LIN {X 0,Y 460.804,Z 363.083,A -85,B 0,C 180,E1 -7827.377,E2 -7827.377} C_VEL
LIN {X 0,Y 460.857,Z 363.08,A -85,B 0,C 180,E1 -7830,E2 -7830} C_VEL
LIN {X 0,Y 460.828,Z 363.084,A -85,B 0,C 180,E1 -7832.622,E2 -7832.622} C_VEL
LIN {X 0,Y 460.706,Z 363.1,A -85,B 0,C 180,E1 -7836.13,E2 -7836.13} C_VEL
LIN {X 0,Y 460.632,Z 363.104,A -85,B 0,C 180,E1 -7838.776,E2 -7838.776} C_VEL
LIN {X 0,Y 460.617,Z 363.109,A -85,B 0,C 180,E1 -7842.445,E2 -7842.445} C_VEL
LIN {X 0,Y 460.604,Z 363.112,A -85,B 0,C 180,E1 -7845.997,E2 -7845.997} C_VEL
LIN {X 0,Y 460.575,Z 363.112,A -85,B 0,C 180,E1 -7848.902,E2 -7848.902} C_VEL
LIN {X 0,Y 460.519,Z 363.124,A -85,B 0,C 180,E1 -7851.485,E2 -7851.485} C_VEL
LIN {X 0,Y 460.545,Z 363.119,A -85,B 0,C 180,E1 -7854.332,E2 -7854.332} C_VEL
LIN {X 0,Y 460.583,Z 363.112,A -85,B 0,C 180,E1 -7857.243,E2 -7857.243} C_VEL
LIN {X 0,Y 460.514,Z 363.119,A -85,B 0,C 180,E1 -7860.24,E2 -7860.24} C_VEL
LIN {X 0,Y 460.532,Z 363.121,A -85,B 0,C 180,E1 -7863.325,E2 -7863.325} C_VEL
LIN {X 0,Y 460.479,Z 363.127,A -85,B 0,C 180,E1 -7866.529,E2 -7866.529} C_VEL
LIN {X 0,Y 460.561,Z 363.116,A -85,B 0,C 180,E1 -7869.859,E2 -7869.859} C_VEL
LIN {X 0,Y 460.516,Z 363.122,A -85,B 0,C 180,E1 -7872.9,E2 -7872.9} C_VEL
LIN {X 0,Y 460.514,Z 363.122,A -85,B 0,C 180,E1 -7875.83,E2 -7875.83} C_VEL
LIN {X 0,Y 460.533,Z 363.119,A -85,B 0,C 180,E1 -7878.989,E2 -7878.989} C_VEL
LIN {X 0,Y 460.529,Z 363.123,A -85,B 0,C 180,E1 -7881.267,E2 -7881.267} C_VEL
LIN {X 0,Y 460.513,Z 363.122,A -85,B 0,C 180,E1 -7884.554,E2 -7884.554} C_VEL
LIN {X 0,Y 460.534,Z 363.12,A -85,B 0,C 180,E1 -7887.716,E2 -7887.716} C_VEL
LIN {X 0,Y 460.543,Z 363.118,A -85,B 0,C 180,E1 -7890.769,E2 -7890.769} C_VEL
LIN {X 0,Y 460.566,Z 363.112,A -85,B 0,C 180,E1 -7893.735,E2 -7893.735} C_VEL
LIN {X 0,Y 460.549,Z 363.12,A -85,B 0,C 180,E1 -7896.624,E2 -7896.624} C_VEL
LIN {X 0,Y 460.555,Z 363.118,A -85,B 0,C 180,E1 -7899.453,E2 -7899.453} C_VEL
LIN {X 0,Y 460.562,Z 363.114,A -85,B 0,C 180,E1 -7902.23,E2 -7902.23} C_VEL
LIN {X 0,Y 460.568,Z 363.116,A -85,B 0,C 180,E1 -7904.965,E2 -7904.965} C_VEL
LIN {X 0,Y 460.633,Z 363.106,A -85,B 0,C 180,E1 -7907.666,E2 -7907.666} C_VEL
LIN {X 0,Y 460.632,Z 363.109,A -85,B 0,C 180,E1 -7911.224,E2 -7911.224} C_VEL
LIN {X 0,Y 460.713,Z 363.095,A -85,B 0,C 180,E1 -7913.87,E2 -7913.87} C_VEL
LIN {X 0,Y 460.803,Z 363.084,A -85,B 0,C 180,E1 -7917.377,E2 -7917.377} C_VEL
LIN {X 0,Y 460.857,Z 363.081,A -85,B 0,C 180,E1 -7920,E2 -7920} C_VEL
LIN {X 0,Y 460.827,Z 363.083,A -85,B 0,C 180,E1 -7922.622,E2 -7922.622} C_VEL
LIN {X 0,Y 460.712,Z 363.097,A -85,B 0,C 180,E1 -7926.13,E2 -7926.13} C_VEL
LIN {X 0,Y 460.631,Z 363.106,A -85,B 0,C 180,E1 -7928.776,E2 -7928.776} C_VEL
LIN {X 0,Y 460.616,Z 363.109,A -85,B 0,C 180,E1 -7932.445,E2 -7932.445} C_VEL
LIN {X 0,Y 460.602,Z 363.11,A -85,B 0,C 180,E1 -7935.997,E2 -7935.997} C_VEL
LIN {X 0,Y 460.571,Z 363.114,A -85,B 0,C 180,E1 -7939.615,E2 -7939.615} C_VEL
LIN {X 0,Y 460.513,Z 363.121,A -85,B 0,C 180,E1 -7942.429,E2 -7942.429} C_VEL
LIN {X 0,Y 460.57,Z 363.114,A -85,B 0,C 180,E1 -7945.802,E2 -7945.802} C_VEL
LIN {X 0,Y 460.554,Z 363.118,A -85,B 0,C 180,E1 -7948.233,E2 -7948.233} C_VEL
LIN {X 0,Y 460.523,Z 363.12,A -85,B 0,C 180,E1 -7951.283,E2 -7951.283} C_VEL
LIN {X 0,Y 460.536,Z 363.121,A -85,B 0,C 180,E1 -7954.506,E2 -7954.506} C_VEL
LIN {X 0,Y 460.53,Z 363.119,A -85,B 0,C 180,E1 -7957.62,E2 -7957.62} C_VEL
LIN {X 0,Y 460.545,Z 363.117,A -85,B 0,C 180,E1 -7960.27,E2 -7960.27} C_VEL
LIN {X 0,Y 460.511,Z 363.125,A -85,B 0,C 180,E1 -7963.374,E2 -7963.374} C_VEL
LIN {X 0,Y 460.511,Z 363.122,A -85,B 0,C 180,E1 -7966.626,E2 -7966.626} C_VEL
LIN {X 0,Y 460.542,Z 363.121,A -85,B 0,C 180,E1 -7969.731,E2 -7969.731} C_VEL
LIN {X 0,Y 460.501,Z 363.121,A -85,B 0,C 180,E1 -7972.524,E2 -7972.524} C_VEL
LIN {X 0,Y 460.548,Z 363.115,A -85,B 0,C 180,E1 -7975.624,E2 -7975.624} C_VEL
LIN {X 0,Y 460.613,Z 363.263,A -85,B 0,C 180,E1 -7976.739,E2 -7976.739} C_VEL
LIN {X 0,Y 463.241,Z 375.686,A -85,B 0,C 180,E1 -7979.857,E2 -7979.857} C_VEL
LIN {X 0,Y 464.177,Z 380.491,A -85,B 0,C 180,E1 -7981.02,E2 -7981.02} C_VEL
LIN {X 0,Y 463.73,Z 388.112,A -85,B 0,C 180,E1 -7982.713,E2 -7982.713} C_VEL
LIN {X 0,Y 462.742,Z 402.3,A -85,B 0,C 180,E1 -7985.791,E2 -7985.791} C_VEL
LIN {X 0,Y 461.732,Z 418.733,A -85,B 0,C 180,E1 -7989.275,E2 -7989.275} C_VEL
LIN {X 0,Y 461.049,Z 434.161,A -85,B 0,C 180,E1 -7992.479,E2 -7992.479} C_VEL
LIN {X 0,Y 460.614,Z 445.332,A -85,B 0,C 180,E1 -7994.768,E2 -7994.768} C_VEL
LIN {X 0,Y 462.065,Z 459.581,A -85,B 0,C 180,E1 -7995.156,E2 -7995.156} C_VEL
LIN {X 0,Y 462.428,Z 464.556,A -85,B 0,C 180,E1 -7995.336,E2 -7995.336} C_VEL
LIN {X 0,Y 462.148,Z 476.548,A -85,B 0,C 180,E1 -7995.862,E2 -7995.862} C_VEL
LIN {X 0,Y 461.723,Z 488.674,A -85,B 0,C 180,E1 -7996.578,E2 -7996.578} C_VEL
LIN {X 0,Y 461.341,Z 499.812,A -85,B 0,C 180,E1 -7997.428,E2 -7997.428} C_VEL
LIN {X 0,Y 460.794,Z 510.557,A -85,B 0,C 180,E1 -7998.452,E2 -7998.452} C_VEL
LIN {X 0,Y 460.459,Z 519.001,A -85,B 0,C 180,E1 -7999.446,E2 -7999.446} C_VEL
LIN {X 0,Y 460.111,Z 528.13,A -85,B 0,C 180,E1 -8000.771,E2 -8000.771} C_VEL
LIN {X 0,Y 459.892,Z 535.454,A -85,B 0,C 180,E1 -8002.095,E2 -8002.095} C_VEL
LIN {X 0,Y 459.735,Z 541.743,A -85,B 0,C 180,E1 -8003.546,E2 -8003.546} C_VEL
LIN {X 0,Y 459.728,Z 545.798,A -85,B 0,C 180,E1 -8004.737,E2 -8004.737} C_VEL
LIN {X 0,Y 459.681,Z 548.168,A -85,B 0,C 180,E1 -8005.616,E2 -8005.616} C_VEL
LIN {X 0,Y 459.745,Z 550.103,A -85,B 0,C 180,E1 -8006.494,E2 -8006.494} C_VEL
LIN {X 0,Y 459.762,Z 551.576,A -85,B 0,C 180,E1 -8007.372,E2 -8007.372} C_VEL
LIN {X 0,Y 459.6,Z 553.186,A -85,B 0,C 180,E1 -8009.124,E2 -8009.124} C_VEL
LIN {X 0,Y 459.605,Z 553.392,A -85,B 0,C 180,E1 -8010,E2 -8010} C_VEL
LIN {X 0,Y 459.603,Z 553.142,A -85,B 0,C 180,E1 -8010.876,E2 -8010.876} C_VEL
LIN {X 0,Y 459.765,Z 551.428,A -85,B 0,C 180,E1 -8012.628,E2 -8012.628} C_VEL
LIN {X 0,Y 459.759,Z 549.92,A -85,B 0,C 180,E1 -8013.506,E2 -8013.506} C_VEL
LIN {X 0,Y 459.668,Z 546.785,A -85,B 0,C 180,E1 -8014.824,E2 -8014.824} C_VEL
LIN {X 0,Y 459.757,Z 542.559,A -85,B 0,C 180,E1 -8016.143,E2 -8016.143} C_VEL
LIN {X 0,Y 459.854,Z 537.104,A -85,B 0,C 180,E1 -8017.464,E2 -8017.464} C_VEL
LIN {X 0,Y 460.018,Z 530.243,A -85,B 0,C 180,E1 -8018.788,E2 -8018.788} C_VEL
LIN {X 0,Y 460.303,Z 521.708,A -85,B 0,C 180,E1 -8020.113,E2 -8020.113} C_VEL
LIN {X 0,Y 460.698,Z 512.901,A -85,B 0,C 180,E1 -8021.216,E2 -8021.216} C_VEL
LIN {X 0,Y 461.092,Z 503.223,A -85,B 0,C 180,E1 -8022.209,E2 -8022.209} C_VEL
LIN {X 0,Y 461.542,Z 492.388,A -85,B 0,C 180,E1 -8023.112,E2 -8023.112} C_VEL
LIN {X 0,Y 461.963,Z 480.948,A -85,B 0,C 180,E1 -8023.864,E2 -8023.864} C_VEL
LIN {X 0,Y 462.412,Z 467.554,A -85,B 0,C 180,E1 -8024.524,E2 -8024.524} C_VEL
LIN {X 0,Y 462.324,Z 461.772,A -85,B 0,C 180,E1 -8024.751,E2 -8024.751} C_VEL
LIN {X 0,Y 461.146,Z 449.381,A -85,B 0,C 180,E1 -8025.143,E2 -8025.143} C_VEL
LIN {X 0,Y 460.603,Z 444.609,A -85,B 0,C 180,E1 -8025.26,E2 -8025.26} C_VEL
LIN {X 0,Y 461.149,Z 429.066,A -85,B 0,C 180,E1 -8028.435,E2 -8028.435} C_VEL
LIN {X 0,Y 461.893,Z 415.007,A -85,B 0,C 180,E1 -8031.419,E2 -8031.419} C_VEL
LIN {X 0,Y 462.96,Z 400.561,A -85,B 0,C 180,E1 -8034.674,E2 -8034.674} C_VEL
LIN {X 0,Y 464.43,Z 386.973,A -85,B 0,C 180,E1 -8037.977,E2 -8037.977} C_VEL
LIN {X 0,Y 464.771,Z 383.328,A -85,B 0,C 180,E1 -8038.94,E2 -8038.94} C_VEL
LIN {X 0,Y 463.986,Z 377.841,A -85,B 0,C 180,E1 -8040.594,E2 -8040.594} C_VEL
LIN {X 0,Y 462.269,Z 370.242,A -85,B 0,C 180,E1 -8043.261,E2 -8043.261} C_VEL
LIN {X 0,Y 461.021,Z 365.258,A -85,B 0,C 180,E1 -8045.401,E2 -8045.401} C_VEL
LIN {X 0,Y 460.479,Z 363.13,A -85,B 0,C 180,E1 -8046.529,E2 -8046.529} C_VEL
LIN {X 0,Y 460.535,Z 363.121,A -85,B 0,C 180,E1 -8049.862,E2 -8049.862} C_VEL
LIN {X 0,Y 460.52,Z 363.124,A -85,B 0,C 180,E1 -8052.901,E2 -8052.901} C_VEL
LIN {X 0,Y 460.522,Z 363.123,A -85,B 0,C 180,E1 -8055.829,E2 -8055.829} C_VEL
LIN {X 0,Y 460.544,Z 363.12,A -85,B 0,C 180,E1 -8058.99,E2 -8058.99} C_VEL
LIN {X 0,Y 460.55,Z 363.12,A -85,B 0,C 180,E1 -8061.269,E2 -8061.269} C_VEL
LIN {X 0,Y 460.516,Z 363.125,A -85,B 0,C 180,E1 -8064.555,E2 -8064.555} C_VEL
LIN {X 0,Y 460.57,Z 363.243,A -85,B 0,C 180,E1 -8065.626,E2 -8065.626} C_VEL
LIN {X 0,Y 461.132,Z 366.331,A -85,B 0,C 180,E1 -8067.763,E2 -8067.763} C_VEL
LIN {X 0,Y 461.472,Z 370.302,A -85,B 0,C 180,E1 -8070.237,E2 -8070.237} C_VEL
LIN {X 0,Y 461.266,Z 374.775,A -85,B 0,C 180,E1 -8072.8,E2 -8072.8} C_VEL
LIN {X 0,Y 460.953,Z 380,A -85,B 0,C 180,E1 -8075.691,E2 -8075.691} C_VEL
LIN {X 0,Y 460.78,Z 385.295,A -85,B 0,C 180,E1 -8078.527,E2 -8078.527} C_VEL
LIN {X 0,Y 460.589,Z 390.661,A -85,B 0,C 180,E1 -8081.311,E2 -8081.311} C_VEL
LIN {X 0,Y 460.395,Z 396.113,A -85,B 0,C 180,E1 -8084.093,E2 -8084.093} C_VEL
LIN {X 0,Y 460.212,Z 403.49,A -85,B 0,C 180,E1 -8087.786,E2 -8087.786} C_VEL
LIN {X 0,Y 460.028,Z 408.741,A -85,B 0,C 180,E1 -8090.353,E2 -8090.353} C_VEL
LIN {X 0,Y 461.717,Z 418.634,A -85,B 0,C 180,E1 -8090.914,E2 -8090.914} C_VEL
LIN {X 0,Y 461.425,Z 428.414,A -85,B 0,C 180,E1 -8091.57,E2 -8091.57} C_VEL
LIN {X 0,Y 461.114,Z 437.441,A -85,B 0,C 180,E1 -8092.382,E2 -8092.382} C_VEL
LIN {X 0,Y 460.834,Z 444.616,A -85,B 0,C 180,E1 -8093.212,E2 -8093.212} C_VEL
LIN {X 0,Y 460.601,Z 450.612,A -85,B 0,C 180,E1 -8094.088,E2 -8094.088} C_VEL
LIN {X 0,Y 460.341,Z 456.412,A -85,B 0,C 180,E1 -8095.183,E2 -8095.183} C_VEL
LIN {X 0,Y 460.304,Z 459.937,A -85,B 0,C 180,E1 -8096.06,E2 -8096.06} C_VEL
LIN {X 0,Y 460.105,Z 462.654,A -85,B 0,C 180,E1 -8096.935,E2 -8096.935} C_VEL
LIN {X 0,Y 459.887,Z 463.739,A -85,B 0,C 180,E1 -8097.372,E2 -8097.372} C_VEL
LIN {X 0,Y 459.78,Z 465.333,A -85,B 0,C 180,E1 -8098.248,E2 -8098.248} C_VEL
LIN {X 0,Y 459.732,Z 466.235,A -85,B 0,C 180,E1 -8099.124,E2 -8099.124} C_VEL
LIN {X 0,Y 459.71,Z 466.468,A -85,B 0,C 180,E1 -8100,E2 -8100} C_VEL
LIN {X 0,Y 459.703,Z 466.034,A -85,B 0,C 180,E1 -8100.876,E2 -8100.876} C_VEL
LIN {X 0,Y 459.727,Z 464.929,A -85,B 0,C 180,E1 -8101.752,E2 -8101.752} C_VEL
LIN {X 0,Y 460.036,Z 461.941,A -85,B 0,C 180,E1 -8103.065,E2 -8103.065} C_VEL
LIN {X 0,Y 460.22,Z 457.216,A -85,B 0,C 180,E1 -8104.379,E2 -8104.379} C_VEL
LIN {X 0,Y 460.371,Z 451.718,A -85,B 0,C 180,E1 -8105.475,E2 -8105.475} C_VEL
LIN {X 0,Y 460.495,Z 446.043,A -85,B 0,C 180,E1 -8106.353,E2 -8106.353} C_VEL
LIN {X 0,Y 460.645,Z 438.702,A -85,B 0,C 180,E1 -8107.247,E2 -8107.247} C_VEL
LIN {X 0,Y 460.944,Z 429.462,A -85,B 0,C 180,E1 -8108.108,E2 -8108.108} C_VEL
LIN {X 0,Y 461.224,Z 420.011,A -85,B 0,C 180,E1 -8108.765,E2 -8108.765} C_VEL
LIN {X 0,Y 461.037,Z 415.021,A -85,B 0,C 180,E1 -8109.045,E2 -8109.045} C_VEL
LIN {X 0,Y 459.779,Z 406.698,A -85,B 0,C 180,E1 -8109.458,E2 -8109.458} C_VEL
LIN {X 0,Y 459.856,Z 400.472,A -85,B 0,C 180,E1 -8112.355,E2 -8112.355} C_VEL
LIN {X 0,Y 460.013,Z 392.824,A -85,B 0,C 180,E1 -8115.962,E2 -8115.962} C_VEL
LIN {X 0,Y 460.143,Z 387.009,A -85,B 0,C 180,E1 -8118.744,E2 -8118.744} C_VEL
LIN {X 0,Y 460.21,Z 381.312,A -85,B 0,C 180,E1 -8121.501,E2 -8121.501} C_VEL
LIN {X 0,Y 460.342,Z 375.512,A -85,B 0,C 180,E1 -8124.344,E2 -8124.344} C_VEL
LIN {X 0,Y 460.491,Z 369.662,A -85,B 0,C 180,E1 -8127.249,E2 -8127.249} C_VEL
LIN {X 0,Y 460.777,Z 363.737,A -85,B 0,C 180,E1 -8130.221,E2 -8130.221} C_VEL
LIN {X 0,Y 460.664,Z 363.105,A -85,B 0,C 180,E1 -8130.609,E2 -8130.609} C_VEL
LIN {X 0,Y 460.552,Z 363.117,A -85,B 0,C 180,E1 -8134.376,E2 -8134.376} C_VEL
LIN {X 0,Y 460.532,Z 363.12,A -85,B 0,C 180,E1 -8137.621,E2 -8137.621} C_VEL
LIN {X 0,Y 460.545,Z 363.117,A -85,B 0,C 180,E1 -8140.269,E2 -8140.269} C_VEL
LIN {X 0,Y 460.503,Z 363.121,A -85,B 0,C 180,E1 -8143.375,E2 -8143.375} C_VEL
LIN {X 0,Y 460.512,Z 363.123,A -85,B 0,C 180,E1 -8146.626,E2 -8146.626} C_VEL
LIN {X 0,Y 460.546,Z 363.118,A -85,B 0,C 180,E1 -8149.73,E2 -8149.73} C_VEL
LIN {X 0,Y 460.503,Z 363.123,A -85,B 0,C 180,E1 -8152.524,E2 -8152.524} C_VEL
LIN {X 0,Y 460.549,Z 363.115,A -85,B 0,C 180,E1 -8155.624,E2 -8155.624} C_VEL
LIN {X 0,Y 460.541,Z 363.118,A -85,B 0,C 180,E1 -8158.745,E2 -8158.745} C_VEL
LIN {X 0,Y 460.592,Z 363.111,A -85,B 0,C 180,E1 -8162.252,E2 -8162.252} C_VEL
LIN {X 0,Y 460.535,Z 363.116,A -85,B 0,C 180,E1 -8165.667,E2 -8165.667} C_VEL
LIN {X 0,Y 460.525,Z 363.12,A -85,B 0,C 180,E1 -8168.578,E2 -8168.578} C_VEL
LIN {X 0,Y 460.594,Z 363.112,A -85,B 0,C 180,E1 -8171.311,E2 -8171.311} C_VEL
LIN {X 0,Y 460.571,Z 363.112,A -85,B 0,C 180,E1 -8174.586,E2 -8174.586} C_VEL
LIN {X 0,Y 460.613,Z 363.108,A -85,B 0,C 180,E1 -8177.666,E2 -8177.666} C_VEL
LIN {X 0,Y 460.606,Z 363.108,A -85,B 0,C 180,E1 -8178.39,E2 -8178.39} C_VEL
LIN {X 0,Y 459.966,Z 363.191,A -85,B 0,C 180,E1 -8179.12,E2 -8179.12} C_VEL
LIN {X 0,Y 457.128,Z 363.545,A -85,B 0,C 180,E1 -8180.306,E2 -8180.306} C_VEL
LIN {X 0,Y 454.734,Z 363.842,A -85,B 0,C 180,E1 -8181.262,E2 -8181.262} C_VEL
LIN {X 0,Y 453.735,Z 363.966,A -85,B 0,C 180,E1 -8182.001,E2 -8182.001} C_VEL
LIN {X 0,Y 453.671,Z 363.974,A -85,B 0,C 180,E1 -8182.251,E2 -8182.251} C_VEL
LIN {X 0,Y 453.672,Z 363.975,A -85,B 0,C 180,E1 -8184.667,E2 -8184.667} C_VEL
LIN {X 0,Y 453.748,Z 363.962,A -85,B 0,C 180,E1 -8187.337,E2 -8187.337} C_VEL
LIN {X 0,Y 453.827,Z 363.956,A -85,B 0,C 180,E1 -8190,E2 -8190} C_VEL
LIN {X 0,Y 453.769,Z 363.963,A -85,B 0,C 180,E1 -8192.663,E2 -8192.663} C_VEL
LIN {X 0,Y 453.673,Z 363.976,A -85,B 0,C 180,E1 -8196.225,E2 -8196.225} C_VEL
LIN {X 0,Y 453.596,Z 363.98,A -85,B 0,C 180,E1 -8198.913,E2 -8198.913} C_VEL
LIN {X 0,Y 453.567,Z 363.987,A -85,B 0,C 180,E1 -8202.529,E2 -8202.529} C_VEL
LIN {X 0,Y 453.548,Z 363.991,A -85,B 0,C 180,E1 -8206.196,E2 -8206.196} C_VEL
LIN {X 0,Y 453.524,Z 363.99,A -85,B 0,C 180,E1 -8209.041,E2 -8209.041} C_VEL
LIN {X 0,Y 453.48,Z 363.998,A -85,B 0,C 180,E1 -8211.836,E2 -8211.836} C_VEL
LIN {X 0,Y 453.517,Z 363.994,A -85,B 0,C 180,E1 -8214.734,E2 -8214.734} C_VEL
LIN {X 0,Y 453.541,Z 363.992,A -85,B 0,C 180,E1 -8217.961,E2 -8217.961} C_VEL
LIN {X 0,Y 453.469,Z 364.001,A -85,B 0,C 180,E1 -8221.525,E2 -8221.525} C_VEL
LIN {X 0,Y 453.49,Z 363.997,A -85,B 0,C 180,E1 -8224.777,E2 -8224.777} C_VEL
LIN {X 0,Y 453.467,Z 363.999,A -85,B 0,C 180,E1 -8228.311,E2 -8228.311} C_VEL
LIN {X 0,Y 453.497,Z 363.994,A -85,B 0,C 180,E1 -8230.609,E2 -8230.609} C_VEL
LIN {X 0,Y 453.459,Z 364.003,A -85,B 0,C 180,E1 -8233.244,E2 -8233.244} C_VEL
LIN {X 0,Y 453.469,Z 363.999,A -85,B 0,C 180,E1 -8235.779,E2 -8235.779} C_VEL
LIN {X 0,Y 453.481,Z 363.998,A -85,B 0,C 180,E1 -8238.209,E2 -8238.209} C_VEL
LIN {X 0,Y 453.497,Z 363.995,A -85,B 0,C 180,E1 -8240.793,E2 -8240.793} C_VEL
LIN {X 0,Y 453.457,Z 363.999,A -85,B 0,C 180,E1 -8243.917,E2 -8243.917} C_VEL
LIN {X 0,Y 453.485,Z 363.997,A -85,B 0,C 180,E1 -8247.151,E2 -8247.151} C_VEL
LIN {X 0,Y 453.478,Z 363.998,A -85,B 0,C 180,E1 -8250.268,E2 -8250.268} C_VEL
LIN {X 0,Y 453.509,Z 363.994,A -85,B 0,C 180,E1 -8253.294,E2 -8253.294} C_VEL
LIN {X 0,Y 453.507,Z 363.994,A -85,B 0,C 180,E1 -8256.239,E2 -8256.239} C_VEL
LIN {X 0,Y 453.486,Z 363.997,A -85,B 0,C 180,E1 -8259.118,E2 -8259.118} C_VEL
LIN {X 0,Y 453.515,Z 363.993,A -85,B 0,C 180,E1 -8261.945,E2 -8261.945} C_VEL
LIN {X 0,Y 453.543,Z 363.993,A -85,B 0,C 180,E1 -8264.726,E2 -8264.726} C_VEL
LIN {X 0,Y 453.605,Z 363.982,A -85,B 0,C 180,E1 -8267.472,E2 -8267.472} C_VEL
LIN {X 0,Y 453.596,Z 363.985,A -85,B 0,C 180,E1 -8271.087,E2 -8271.087} C_VEL
LIN {X 0,Y 453.68,Z 363.972,A -85,B 0,C 180,E1 -8273.775,E2 -8273.775} C_VEL
LIN {X 0,Y 453.747,Z 363.963,A -85,B 0,C 180,E1 -8277.337,E2 -8277.337} C_VEL
LIN {X 0,Y 453.827,Z 363.957,A -85,B 0,C 180,E1 -8280,E2 -8280} C_VEL
LIN {X 0,Y 453.768,Z 363.963,A -85,B 0,C 180,E1 -8282.663,E2 -8282.663} C_VEL
LIN {X 0,Y 453.68,Z 363.974,A -85,B 0,C 180,E1 -8286.225,E2 -8286.225} C_VEL
LIN {X 0,Y 453.594,Z 363.982,A -85,B 0,C 180,E1 -8288.913,E2 -8288.913} C_VEL
LIN {X 0,Y 453.566,Z 363.987,A -85,B 0,C 180,E1 -8292.529,E2 -8292.529} C_VEL
LIN {X 0,Y 453.546,Z 363.991,A -85,B 0,C 180,E1 -8296.196,E2 -8296.196} C_VEL
LIN {X 0,Y 453.52,Z 363.991,A -85,B 0,C 180,E1 -8299.04,E2 -8299.04} C_VEL
LIN {X 0,Y 453.478,Z 364,A -85,B 0,C 180,E1 -8301.836,E2 -8301.836} C_VEL
LIN {X 0,Y 453.515,Z 363.994,A -85,B 0,C 180,E1 -8304.734,E2 -8304.734} C_VEL
LIN {X 0,Y 453.534,Z 363.993,A -85,B 0,C 180,E1 -8307.96,E2 -8307.96} C_VEL
LIN {X 0,Y 453.468,Z 364.001,A -85,B 0,C 180,E1 -8311.525,E2 -8311.525} C_VEL
LIN {X 0,Y 453.491,Z 363.997,A -85,B 0,C 180,E1 -8314.778,E2 -8314.778} C_VEL
LIN {X 0,Y 453.475,Z 363.999,A -85,B 0,C 180,E1 -8318.311,E2 -8318.311} C_VEL
LIN {X 0,Y 453.496,Z 363.993,A -85,B 0,C 180,E1 -8320.609,E2 -8320.609} C_VEL
LIN {X 0,Y 453.465,Z 364.001,A -85,B 0,C 180,E1 -8323.245,E2 -8323.245} C_VEL
LIN {X 0,Y 453.475,Z 363.998,A -85,B 0,C 180,E1 -8325.78,E2 -8325.78} C_VEL
LIN {X 0,Y 453.484,Z 363.999,A -85,B 0,C 180,E1 -8328.21,E2 -8328.21} C_VEL
LIN {X 0,Y 453.489,Z 363.992,A -85,B 0,C 180,E1 -8330.794,E2 -8330.794} C_VEL
LIN {X 0,Y 453.456,Z 364.001,A -85,B 0,C 180,E1 -8333.917,E2 -8333.917} C_VEL
LIN {X 0,Y 453.551,Z 364.167,A -85,B 0,C 180,E1 -8336.43,E2 -8336.43} C_VEL
LIN {X 0,Y 456.236,Z 376.608,A -85,B 0,C 180,E1 -8339.615,E2 -8339.615} C_VEL
LIN {X 0,Y 457.29,Z 382.993,A -85,B 0,C 180,E1 -8341.166,E2 -8341.166} C_VEL
LIN {X 0,Y 456.263,Z 396.521,A -85,B 0,C 180,E1 -8344.205,E2 -8344.205} C_VEL
LIN {X 0,Y 455.153,Z 412.385,A -85,B 0,C 180,E1 -8347.665,E2 -8347.665} C_VEL
LIN {X 0,Y 454.34,Z 426.401,A -85,B 0,C 180,E1 -8350.663,E2 -8350.663} C_VEL
LIN {X 0,Y 453.726,Z 440.257,A -85,B 0,C 180,E1 -8353.58,E2 -8353.58} C_VEL
LIN {X 0,Y 453.581,Z 445.076,A -85,B 0,C 180,E1 -8354.585,E2 -8354.585} C_VEL
LIN {X 0,Y 454.967,Z 459.21,A -85,B 0,C 180,E1 -8354.976,E2 -8354.976} C_VEL
LIN {X 0,Y 455.443,Z 464.957,A -85,B 0,C 180,E1 -8355.192,E2 -8355.192} C_VEL
LIN {X 0,Y 455.135,Z 477.261,A -85,B 0,C 180,E1 -8355.753,E2 -8355.753} C_VEL
LIN {X 0,Y 454.693,Z 489.054,A -85,B 0,C 180,E1 -8356.48,E2 -8356.48} C_VEL
LIN {X 0,Y 454.283,Z 500.104,A -85,B 0,C 180,E1 -8357.35,E2 -8357.35} C_VEL
LIN {X 0,Y 453.732,Z 510.602,A -85,B 0,C 180,E1 -8358.383,E2 -8358.383} C_VEL
LIN {X 0,Y 453.326,Z 519.758,A -85,B 0,C 180,E1 -8359.504,E2 -8359.504} C_VEL
LIN {X 0,Y 453.015,Z 528.665,A -85,B 0,C 180,E1 -8360.85,E2 -8360.85} C_VEL
LIN {X 0,Y 452.805,Z 535.733,A -85,B 0,C 180,E1 -8362.195,E2 -8362.195} C_VEL
LIN {X 0,Y 452.65,Z 541.426,A -85,B 0,C 180,E1 -8363.559,E2 -8363.559} C_VEL
LIN {X 0,Y 452.589,Z 546.336,A -85,B 0,C 180,E1 -8365.101,E2 -8365.101} C_VEL
LIN {X 0,Y 452.674,Z 549.413,A -85,B 0,C 180,E1 -8366.44,E2 -8366.44} C_VEL
LIN {X 0,Y 452.706,Z 550.901,A -85,B 0,C 180,E1 -8367.331,E2 -8367.331} C_VEL
LIN {X 0,Y 452.589,Z 551.908,A -85,B 0,C 180,E1 -8368.22,E2 -8368.22} C_VEL
LIN {X 0,Y 452.533,Z 552.516,A -85,B 0,C 180,E1 -8369.11,E2 -8369.11} C_VEL
LIN {X 0,Y 452.536,Z 552.724,A -85,B 0,C 180,E1 -8370,E2 -8370} C_VEL
LIN {X 0,Y 452.536,Z 552.477,A -85,B 0,C 180,E1 -8370.89,E2 -8370.89} C_VEL
LIN {X 0,Y 452.592,Z 551.819,A -85,B 0,C 180,E1 -8371.78,E2 -8371.78} C_VEL
LIN {X 0,Y 452.71,Z 550.759,A -85,B 0,C 180,E1 -8372.669,E2 -8372.669} C_VEL
LIN {X 0,Y 452.654,Z 548.304,A -85,B 0,C 180,E1 -8374.006,E2 -8374.006} C_VEL
LIN {X 0,Y 452.677,Z 544.812,A -85,B 0,C 180,E1 -8375.345,E2 -8375.345} C_VEL
LIN {X 0,Y 452.759,Z 539.621,A -85,B 0,C 180,E1 -8376.832,E2 -8376.832} C_VEL
LIN {X 0,Y 452.882,Z 533.154,A -85,B 0,C 180,E1 -8378.253,E2 -8378.253} C_VEL
LIN {X 0,Y 453.099,Z 525.487,A -85,B 0,C 180,E1 -8379.599,E2 -8379.599} C_VEL
LIN {X 0,Y 453.419,Z 517.654,A -85,B 0,C 180,E1 -8380.72,E2 -8380.72} C_VEL
LIN {X 0,Y 453.861,Z 506.991,A -85,B 0,C 180,E1 -8381.953,E2 -8381.953} C_VEL
LIN {X 0,Y 454.307,Z 496.361,A -85,B 0,C 180,E1 -8382.942,E2 -8382.942} C_VEL
LIN {X 0,Y 454.763,Z 485.534,A -85,B 0,C 180,E1 -8383.746,E2 -8383.746} C_VEL
LIN {X 0,Y 455.326,Z 472.817,A -85,B 0,C 180,E1 -8384.469,E2 -8384.469} C_VEL
LIN {X 0,Y 455.363,Z 462.344,A -85,B 0,C 180,E1 -8384.925,E2 -8384.925} C_VEL
LIN {X 0,Y 454.227,Z 449.851,A -85,B 0,C 180,E1 -8385.347,E2 -8385.347} C_VEL
LIN {X 0,Y 453.567,Z 444.274,A -85,B 0,C 180,E1 -8385.495,E2 -8385.495} C_VEL
LIN {X 0,Y 454.191,Z 428.804,A -85,B 0,C 180,E1 -8388.728,E2 -8388.728} C_VEL
LIN {X 0,Y 454.998,Z 414.943,A -85,B 0,C 180,E1 -8391.76,E2 -8391.76} C_VEL
LIN {X 0,Y 456.14,Z 400.646,A -85,B 0,C 180,E1 -8395.069,E2 -8395.069} C_VEL
LIN {X 0,Y 457.778,Z 387.378,A -85,B 0,C 180,E1 -8398.42,E2 -8398.42} C_VEL
LIN {X 0,Y 457.886,Z 383.82,A -85,B 0,C 180,E1 -8399.417,E2 -8399.417} C_VEL
LIN {X 0,Y 456.615,Z 377.293,A -85,B 0,C 180,E1 -8401.555,E2 -8401.555} C_VEL
LIN {X 0,Y 455.348,Z 371.453,A -85,B 0,C 180,E1 -8403.755,E2 -8403.755} C_VEL
LIN {X 0,Y 454.054,Z 366.532,A -85,B 0,C 180,E1 -8406.028,E2 -8406.028} C_VEL
LIN {X 0,Y 453.471,Z 364.002,A -85,B 0,C 180,E1 -8407.479,E2 -8407.479} C_VEL
LIN {X 0,Y 453.497,Z 363.998,A -85,B 0,C 180,E1 -8410.609,E2 -8410.609} C_VEL
LIN {X 0,Y 453.466,Z 364.002,A -85,B 0,C 180,E1 -8413.245,E2 -8413.245} C_VEL
LIN {X 0,Y 453.476,Z 364.001,A -85,B 0,C 180,E1 -8415.78,E2 -8415.78} C_VEL
LIN {X 0,Y 453.519,Z 363.995,A -85,B 0,C 180,E1 -8419.406,E2 -8419.406} C_VEL
LIN {X 0,Y 453.481,Z 364.001,A -85,B 0,C 180,E1 -8422.223,E2 -8422.223} C_VEL
LIN {X 0,Y 453.476,Z 364.038,A -85,B 0,C 180,E1 -8424.739,E2 -8424.739} C_VEL
LIN {X 0,Y 454.165,Z 367.303,A -85,B 0,C 180,E1 -8427.207,E2 -8427.207} C_VEL
LIN {X 0,Y 454.568,Z 371.516,A -85,B 0,C 180,E1 -8429.975,E2 -8429.975} C_VEL
LIN {X 0,Y 454.385,Z 375.522,A -85,B 0,C 180,E1 -8432.354,E2 -8432.354} C_VEL
LIN {X 0,Y 454.023,Z 380.711,A -85,B 0,C 180,E1 -8435.295,E2 -8435.295} C_VEL
LIN {X 0,Y 453.8,Z 386.229,A -85,B 0,C 180,E1 -8438.314,E2 -8438.314} C_VEL
LIN {X 0,Y 453.6,Z 391.275,A -85,B 0,C 180,E1 -8441.012,E2 -8441.012} C_VEL
LIN {X 0,Y 453.391,Z 396.966,A -85,B 0,C 180,E1 -8443.959,E2 -8443.959} C_VEL
LIN {X 0,Y 453.183,Z 404.321,A -85,B 0,C 180,E1 -8447.692,E2 -8447.692} C_VEL
LIN {X 0,Y 452.982,Z 409.199,A -85,B 0,C 180,E1 -8450.117,E2 -8450.117} C_VEL
LIN {X 0,Y 454.751,Z 418.551,A -85,B 0,C 180,E1 -8450.661,E2 -8450.661} C_VEL
LIN {X 0,Y 454.645,Z 426.986,A -85,B 0,C 180,E1 -8451.22,E2 -8451.22} C_VEL
LIN {X 0,Y 454.327,Z 436.017,A -85,B 0,C 180,E1 -8451.997,E2 -8451.997} C_VEL
LIN {X 0,Y 453.955,Z 443.972,A -85,B 0,C 180,E1 -8452.885,E2 -8452.885} C_VEL
LIN {X 0,Y 453.626,Z 450.223,A -85,B 0,C 180,E1 -8453.774,E2 -8453.774} C_VEL
LIN {X 0,Y 453.365,Z 456.268,A -85,B 0,C 180,E1 -8454.886,E2 -8454.886} C_VEL
LIN {X 0,Y 453.278,Z 460.745,A -85,B 0,C 180,E1 -8455.999,E2 -8455.999} C_VEL
LIN {X 0,Y 453.069,Z 463.435,A -85,B 0,C 180,E1 -8456.888,E2 -8456.888} C_VEL
LIN {X 0,Y 452.837,Z 464.508,A -85,B 0,C 180,E1 -8457.331,E2 -8457.331} C_VEL
LIN {X 0,Y 452.724,Z 466.078,A -85,B 0,C 180,E1 -8458.221,E2 -8458.221} C_VEL
LIN {X 0,Y 452.67,Z 466.955,A -85,B 0,C 180,E1 -8459.11,E2 -8459.11} C_VEL
LIN {X 0,Y 452.645,Z 467.162,A -85,B 0,C 180,E1 -8460,E2 -8460} C_VEL
LIN {X 0,Y 452.636,Z 466.7,A -85,B 0,C 180,E1 -8460.89,E2 -8460.89} C_VEL
LIN {X 0,Y 452.664,Z 465.565,A -85,B 0,C 180,E1 -8461.78,E2 -8461.78} C_VEL
LIN {X 0,Y 452.972,Z 462.529,A -85,B 0,C 180,E1 -8463.113,E2 -8463.113} C_VEL
LIN {X 0,Y 453.168,Z 457.752,A -85,B 0,C 180,E1 -8464.447,E2 -8464.447} C_VEL
LIN {X 0,Y 453.343,Z 452.204,A -85,B 0,C 180,E1 -8465.56,E2 -8465.56} C_VEL
LIN {X 0,Y 453.461,Z 444.834,A -85,B 0,C 180,E1 -8466.675,E2 -8466.675} C_VEL
LIN {X 0,Y 453.723,Z 437.322,A -85,B 0,C 180,E1 -8467.546,E2 -8467.546} C_VEL
LIN {X 0,Y 453.958,Z 428.414,A -85,B 0,C 180,E1 -8468.345,E2 -8468.345} C_VEL
LIN {X 0,Y 454.265,Z 418.463,A -85,B 0,C 180,E1 -8469.012,E2 -8469.012} C_VEL
LIN {X 0,Y 453.026,Z 409.304,A -85,B 0,C 180,E1 -8469.487,E2 -8469.487} C_VEL
LIN {X 0,Y 452.713,Z 406.981,A -85,B 0,C 180,E1 -8469.607,E2 -8469.607} C_VEL
LIN {X 0,Y 452.782,Z 400.713,A -85,B 0,C 180,E1 -8472.551,E2 -8472.551} C_VEL
LIN {X 0,Y 452.969,Z 393.76,A -85,B 0,C 180,E1 -8475.854,E2 -8475.854} C_VEL
LIN {X 0,Y 453.069,Z 387.215,A -85,B 0,C 180,E1 -8479.011,E2 -8479.011} C_VEL
LIN {X 0,Y 453.16,Z 381.408,A -85,B 0,C 180,E1 -8481.852,E2 -8481.852} C_VEL
LIN {X 0,Y 453.317,Z 375.572,A -85,B 0,C 180,E1 -8484.746,E2 -8484.746} C_VEL
LIN {X 0,Y 453.519,Z 369.186,A -85,B 0,C 180,E1 -8487.956,E2 -8487.956} C_VEL
LIN {X 0,Y 453.652,Z 364.015,A -85,B 0,C 180,E1 -8490.59,E2 -8490.59} C_VEL
LIN {X 0,Y 453.482,Z 363.995,A -85,B 0,C 180,E1 -8493.913,E2 -8493.913} C_VEL
LIN {X 0,Y 453.474,Z 363.998,A -85,B 0,C 180,E1 -8497.188,E2 -8497.188} C_VEL
LIN {X 0,Y 453.509,Z 363.995,A -85,B 0,C 180,E1 -8499.448,E2 -8499.448} C_VEL
LIN {X 0,Y 453.467,Z 364.001,A -85,B 0,C 180,E1 -8502.995,E2 -8502.995} C_VEL
LIN {X 0,Y 453.477,Z 363.997,A -85,B 0,C 180,E1 -8505.78,E2 -8505.78} C_VEL
LIN {X 0,Y 453.485,Z 363.999,A -85,B 0,C 180,E1 -8508.21,E2 -8508.21} C_VEL
LIN {X 0,Y 453.498,Z 363.996,A -85,B 0,C 180,E1 -8510.793,E2 -8510.793} C_VEL
LIN {X 0,Y 453.458,Z 363.998,A -85,B 0,C 180,E1 -8513.917,E2 -8513.917} C_VEL
LIN {X 0,Y 453.487,Z 363.996,A -85,B 0,C 180,E1 -8517.151,E2 -8517.151} C_VEL
LIN {X 0,Y 453.479,Z 363.998,A -85,B 0,C 180,E1 -8520.268,E2 -8520.268} C_VEL
LIN {X 0,Y 453.509,Z 363.993,A -85,B 0,C 180,E1 -8523.294,E2 -8523.294} C_VEL
LIN {X 0,Y 453.502,Z 363.997,A -85,B 0,C 180,E1 -8526.239,E2 -8526.239} C_VEL
LIN {X 0,Y 453.486,Z 363.997,A -85,B 0,C 180,E1 -8529.118,E2 -8529.118} C_VEL
LIN {X 0,Y 453.515,Z 363.994,A -85,B 0,C 180,E1 -8531.945,E2 -8531.945} C_VEL
LIN {X 0,Y 453.544,Z 363.991,A -85,B 0,C 180,E1 -8534.726,E2 -8534.726} C_VEL
LIN {X 0,Y 453.564,Z 363.988,A -85,B 0,C 180,E1 -8538.38,E2 -8538.38} C_VEL
LIN {X 0,Y 453.656,Z 363.976,A -85,B 0,C 180,E1 -8541.985,E2 -8541.985} C_VEL
LIN {X 0,Y 453.671,Z 363.974,A -85,B 0,C 180,E1 -8542.251,E2 -8542.251} C_VEL
LIN {X 0,Y 453.025,Z 364.056,A -85,B 0,C 180,E1 -8542.992,E2 -8542.992} C_VEL
LIN {X 0,Y 450.092,Z 364.421,A -85,B 0,C 180,E1 -8544.194,E2 -8544.194} C_VEL
LIN {X 0,Y 447.597,Z 364.73,A -85,B 0,C 180,E1 -8545.165,E2 -8545.165} C_VEL
LIN {X 0,Y 446.542,Z 364.862,A -85,B 0,C 180,E1 -8545.916,E2 -8545.916} C_VEL
LIN {X 0,Y 446.467,Z 364.871,A -85,B 0,C 180,E1 -8546.17,E2 -8546.17} C_VEL
LIN {X 0,Y 446.668,Z 364.848,A -85,B 0,C 180,E1 -8548.197,E2 -8548.197} C_VEL
LIN {X 0,Y 446.797,Z 364.832,A -85,B 0,C 180,E1 -8550,E2 -8550} C_VEL
LIN {X 0,Y 446.712,Z 364.841,A -85,B 0,C 180,E1 -8552.705,E2 -8552.705} C_VEL
LIN {X 0,Y 446.643,Z 364.851,A -85,B 0,C 180,E1 -8556.324,E2 -8556.324} C_VEL
LIN {X 0,Y 446.542,Z 364.859,A -85,B 0,C 180,E1 -8559.055,E2 -8559.055} C_VEL
LIN {X 0,Y 446.525,Z 364.864,A -85,B 0,C 180,E1 -8562.73,E2 -8562.73} C_VEL
LIN {X 0,Y 446.5,Z 364.869,A -85,B 0,C 180,E1 -8566.228,E2 -8566.228} C_VEL
LIN {X 0,Y 446.473,Z 364.87,A -85,B 0,C 180,E1 -8569.303,E2 -8569.303} C_VEL
LIN {X 0,Y 446.421,Z 364.876,A -85,B 0,C 180,E1 -8572.199,E2 -8572.199} C_VEL
LIN {X 0,Y 446.461,Z 364.873,A -85,B 0,C 180,E1 -8575.152,E2 -8575.152} C_VEL
LIN {X 0,Y 446.488,Z 364.869,A -85,B 0,C 180,E1 -8578.178,E2 -8578.178} C_VEL
LIN {X 0,Y 446.423,Z 364.877,A -85,B 0,C 180,E1 -8581.775,E2 -8581.775} C_VEL
LIN {X 0,Y 446.432,Z 364.875,A -85,B 0,C 180,E1 -8584.523,E2 -8584.523} C_VEL
LIN {X 0,Y 446.419,Z 364.878,A -85,B 0,C 180,E1 -8588.079,E2 -8588.079} C_VEL
LIN {X 0,Y 446.43,Z 364.875,A -85,B 0,C 180,E1 -8590.918,E2 -8590.918} C_VEL
LIN {X 0,Y 446.405,Z 364.878,A -85,B 0,C 180,E1 -8593.846,E2 -8593.846} C_VEL
LIN {X 0,Y 446.402,Z 364.88,A -85,B 0,C 180,E1 -8596.403,E2 -8596.403} C_VEL
LIN {X 0,Y 446.429,Z 364.876,A -85,B 0,C 180,E1 -8599.082,E2 -8599.082} C_VEL
LIN {X 0,Y 446.412,Z 364.876,A -85,B 0,C 180,E1 -8602.121,E2 -8602.121} C_VEL
LIN {X 0,Y 446.431,Z 364.875,A -85,B 0,C 180,E1 -8605.477,E2 -8605.477} C_VEL
LIN {X 0,Y 446.418,Z 364.878,A -85,B 0,C 180,E1 -8608.7,E2 -8608.7} C_VEL
LIN {X 0,Y 446.487,Z 364.868,A -85,B 0,C 180,E1 -8611.821,E2 -8611.821} C_VEL
LIN {X 0,Y 446.461,Z 364.875,A -85,B 0,C 180,E1 -8614.848,E2 -8614.848} C_VEL
LIN {X 0,Y 446.451,Z 364.874,A -85,B 0,C 180,E1 -8618.245,E2 -8618.245} C_VEL
LIN {X 0,Y 446.461,Z 364.872,A -85,B 0,C 180,E1 -8621.649,E2 -8621.649} C_VEL
LIN {X 0,Y 446.51,Z 364.866,A -85,B 0,C 180,E1 -8624.48,E2 -8624.48} C_VEL
LIN {X 0,Y 446.542,Z 364.863,A -85,B 0,C 180,E1 -8628.194,E2 -8628.194} C_VEL
LIN {X 0,Y 446.603,Z 364.855,A -85,B 0,C 180,E1 -8631.858,E2 -8631.858} C_VEL
LIN {X 0,Y 446.648,Z 364.851,A -85,B 0,C 180,E1 -8634.583,E2 -8634.583} C_VEL
LIN {X 0,Y 446.667,Z 364.849,A -85,B 0,C 180,E1 -8638.197,E2 -8638.197} C_VEL
LIN {X 0,Y 446.797,Z 364.832,A -85,B 0,C 180,E1 -8640,E2 -8640} C_VEL
LIN {X 0,Y 446.712,Z 364.842,A -85,B 0,C 180,E1 -8642.705,E2 -8642.705} C_VEL
LIN {X 0,Y 446.649,Z 364.851,A -85,B 0,C 180,E1 -8646.324,E2 -8646.324} C_VEL
LIN {X 0,Y 446.54,Z 364.861,A -85,B 0,C 180,E1 -8649.055,E2 -8649.055} C_VEL
LIN {X 0,Y 446.524,Z 364.866,A -85,B 0,C 180,E1 -8652.73,E2 -8652.73} C_VEL
LIN {X 0,Y 446.498,Z 364.869,A -85,B 0,C 180,E1 -8656.228,E2 -8656.228} C_VEL
LIN {X 0,Y 446.471,Z 364.869,A -85,B 0,C 180,E1 -8659.303,E2 -8659.303} C_VEL
LIN {X 0,Y 446.42,Z 364.877,A -85,B 0,C 180,E1 -8662.2,E2 -8662.2} C_VEL
LIN {X 0,Y 446.459,Z 364.872,A -85,B 0,C 180,E1 -8665.152,E2 -8665.152} C_VEL
LIN {X 0,Y 446.486,Z 364.871,A -85,B 0,C 180,E1 -8668.179,E2 -8668.179} C_VEL
LIN {X 0,Y 446.421,Z 364.879,A -85,B 0,C 180,E1 -8671.775,E2 -8671.775} C_VEL
LIN {X 0,Y 446.432,Z 364.877,A -85,B 0,C 180,E1 -8674.523,E2 -8674.523} C_VEL
LIN {X 0,Y 446.433,Z 364.878,A -85,B 0,C 180,E1 -8678.082,E2 -8678.082} C_VEL
LIN {X 0,Y 446.429,Z 364.874,A -85,B 0,C 180,E1 -8680.918,E2 -8680.918} C_VEL
LIN {X 0,Y 446.425,Z 364.877,A -85,B 0,C 180,E1 -8683.843,E2 -8683.843} C_VEL
LIN {X 0,Y 446.423,Z 364.878,A -85,B 0,C 180,E1 -8686.4,E2 -8686.4} C_VEL
LIN {X 0,Y 446.443,Z 364.877,A -85,B 0,C 180,E1 -8689.802,E2 -8689.802} C_VEL
LIN {X 0,Y 446.403,Z 364.882,A -85,B 0,C 180,E1 -8693.255,E2 -8693.255} C_VEL
LIN {X 0,Y 446.516,Z 365.016,A -85,B 0,C 180,E1 -8696.105,E2 -8696.105} C_VEL
LIN {X 0,Y 449.45,Z 378.742,A -85,B 0,C 180,E1 -8699.685,E2 -8699.685} C_VEL
LIN {X 0,Y 450.355,Z 384.304,A -85,B 0,C 180,E1 -8701.068,E2 -8701.068} C_VEL
LIN {X 0,Y 449.338,Z 397.278,A -85,B 0,C 180,E1 -8704.027,E2 -8704.027} C_VEL
LIN {X 0,Y 448.205,Z 412.358,A -85,B 0,C 180,E1 -8707.384,E2 -8707.384} C_VEL
LIN {X 0,Y 447.261,Z 427.703,A -85,B 0,C 180,E1 -8710.732,E2 -8710.732} C_VEL
LIN {X 0,Y 446.643,Z 441.558,A -85,B 0,C 180,E1 -8713.709,E2 -8713.709} C_VEL
LIN {X 0,Y 446.512,Z 444.832,A -85,B 0,C 180,E1 -8714.406,E2 -8714.406} C_VEL
LIN {X 0,Y 447.848,Z 458.556,A -85,B 0,C 180,E1 -8714.79,E2 -8714.79} C_VEL
LIN {X 0,Y 448.451,Z 465.884,A -85,B 0,C 180,E1 -8715.072,E2 -8715.072} C_VEL
LIN {X 0,Y 448.095,Z 478.725,A -85,B 0,C 180,E1 -8715.698,E2 -8715.698} C_VEL
LIN {X 0,Y 447.578,Z 490.758,A -85,B 0,C 180,E1 -8716.482,E2 -8716.482} C_VEL
LIN {X 0,Y 447.175,Z 501.765,A -85,B 0,C 180,E1 -8717.405,E2 -8717.405} C_VEL
LIN {X 0,Y 446.658,Z 511.573,A -85,B 0,C 180,E1 -8718.427,E2 -8718.427} C_VEL
LIN {X 0,Y 446.204,Z 520.476,A -85,B 0,C 180,E1 -8719.564,E2 -8719.564} C_VEL
LIN {X 0,Y 445.946,Z 527.802,A -85,B 0,C 180,E1 -8720.704,E2 -8720.704} C_VEL
LIN {X 0,Y 445.728,Z 534.943,A -85,B 0,C 180,E1 -8722.07,E2 -8722.07} C_VEL
LIN {X 0,Y 445.569,Z 541.076,A -85,B 0,C 180,E1 -8723.569,E2 -8723.569} C_VEL
LIN {X 0,Y 445.525,Z 545.613,A -85,B 0,C 180,E1 -8725.023,E2 -8725.023} C_VEL
LIN {X 0,Y 445.604,Z 548.711,A -85,B 0,C 180,E1 -8726.383,E2 -8726.383} C_VEL
LIN {X 0,Y 445.652,Z 550.216,A -85,B 0,C 180,E1 -8727.288,E2 -8727.288} C_VEL
LIN {X 0,Y 445.532,Z 551.229,A -85,B 0,C 180,E1 -8728.192,E2 -8728.192} C_VEL
LIN {X 0,Y 445.468,Z 551.84,A -85,B 0,C 180,E1 -8729.096,E2 -8729.096} C_VEL
LIN {X 0,Y 445.469,Z 552.053,A -85,B 0,C 180,E1 -8730,E2 -8730} C_VEL
LIN {X 0,Y 445.471,Z 551.811,A -85,B 0,C 180,E1 -8730.904,E2 -8730.904} C_VEL
LIN {X 0,Y 445.535,Z 551.154,A -85,B 0,C 180,E1 -8731.808,E2 -8731.808} C_VEL
LIN {X 0,Y 445.656,Z 550.094,A -85,B 0,C 180,E1 -8732.712,E2 -8732.712} C_VEL
LIN {X 0,Y 445.588,Z 547.637,A -85,B 0,C 180,E1 -8734.07,E2 -8734.07} C_VEL
LIN {X 0,Y 445.615,Z 544.143,A -85,B 0,C 180,E1 -8735.43,E2 -8735.43} C_VEL
LIN {X 0,Y 445.675,Z 538.708,A -85,B 0,C 180,E1 -8736.997,E2 -8736.997} C_VEL
LIN {X 0,Y 445.856,Z 531.316,A -85,B 0,C 180,E1 -8738.612,E2 -8738.612} C_VEL
LIN {X 0,Y 446.059,Z 523.341,A -85,B 0,C 180,E1 -8739.981,E2 -8739.981} C_VEL
LIN {X 0,Y 446.45,Z 515.177,A -85,B 0,C 180,E1 -8741.119,E2 -8741.119} C_VEL
LIN {X 0,Y 446.88,Z 506.288,A -85,B 0,C 180,E1 -8742.143,E2 -8742.143} C_VEL
LIN {X 0,Y 447.297,Z 496.722,A -85,B 0,C 180,E1 -8743.054,E2 -8743.054} C_VEL
LIN {X 0,Y 447.754,Z 486.493,A -85,B 0,C 180,E1 -8743.849,E2 -8743.849} C_VEL
LIN {X 0,Y 448.34,Z 474.345,A -85,B 0,C 180,E1 -8744.584,E2 -8744.584} C_VEL
LIN {X 0,Y 448.451,Z 463.127,A -85,B 0,C 180,E1 -8745.102,E2 -8745.102} C_VEL
LIN {X 0,Y 447.338,Z 450.256,A -85,B 0,C 180,E1 -8745.562,E2 -8745.562} C_VEL
LIN {X 0,Y 446.532,Z 443.857,A -85,B 0,C 180,E1 -8745.756,E2 -8745.756} C_VEL
LIN {X 0,Y 447.228,Z 428.6,A -85,B 0,C 180,E1 -8749.031,E2 -8749.031} C_VEL
LIN {X 0,Y 448.132,Z 414.11,A -85,B 0,C 180,E1 -8752.287,E2 -8752.287} C_VEL
LIN {X 0,Y 449.346,Z 400.843,A -85,B 0,C 180,E1 -8755.475,E2 -8755.475} C_VEL
LIN {X 0,Y 450.864,Z 389.618,A -85,B 0,C 180,E1 -8758.388,E2 -8758.388} C_VEL
LIN {X 0,Y 451.071,Z 385.71,A -85,B 0,C 180,E1 -8759.505,E2 -8759.505} C_VEL
LIN {X 0,Y 449.909,Z 379.6,A -85,B 0,C 180,E1 -8761.554,E2 -8761.554} C_VEL
LIN {X 0,Y 448.631,Z 373.618,A -85,B 0,C 180,E1 -8763.873,E2 -8763.873} C_VEL
LIN {X 0,Y 447.127,Z 367.875,A -85,B 0,C 180,E1 -8766.676,E2 -8766.676} C_VEL
LIN {X 0,Y 446.445,Z 364.877,A -85,B 0,C 180,E1 -8768.64,E2 -8768.64} C_VEL
LIN {X 0,Y 446.432,Z 364.878,A -85,B 0,C 180,E1 -8771.391,E2 -8771.391} C_VEL
LIN {X 0,Y 446.459,Z 364.875,A -85,B 0,C 180,E1 -8774.897,E2 -8774.897} C_VEL
LIN {X 0,Y 446.439,Z 364.877,A -85,B 0,C 180,E1 -8778.61,E2 -8778.61} C_VEL
LIN {X 0,Y 446.478,Z 364.872,A -85,B 0,C 180,E1 -8780.976,E2 -8780.976} C_VEL
LIN {X 0,Y 446.437,Z 364.977,A -85,B 0,C 180,E1 -8783.819,E2 -8783.819} C_VEL
LIN {X 0,Y 447.165,Z 368.373,A -85,B 0,C 180,E1 -8786.627,E2 -8786.627} C_VEL
LIN {X 0,Y 447.542,Z 371.411,A -85,B 0,C 180,E1 -8788.787,E2 -8788.787} C_VEL
LIN {X 0,Y 447.58,Z 374.653,A -85,B 0,C 180,E1 -8790.872,E2 -8790.872} C_VEL
LIN {X 0,Y 447.252,Z 379.72,A -85,B 0,C 180,E1 -8793.897,E2 -8793.897} C_VEL
LIN {X 0,Y 446.92,Z 384.923,A -85,B 0,C 180,E1 -8796.85,E2 -8796.85} C_VEL
LIN {X 0,Y 446.677,Z 390.201,A -85,B 0,C 180,E1 -8799.748,E2 -8799.748} C_VEL
LIN {X 0,Y 446.453,Z 395.525,A -85,B 0,C 180,E1 -8802.597,E2 -8802.597} C_VEL
LIN {X 0,Y 446.21,Z 400.905,A -85,B 0,C 180,E1 -8805.404,E2 -8805.404} C_VEL
LIN {X 0,Y 446.126,Z 406.316,A -85,B 0,C 180,E1 -8808.183,E2 -8808.183} C_VEL
LIN {X 0,Y 445.991,Z 409.693,A -85,B 0,C 180,E1 -8809.875,E2 -8809.875} C_VEL
LIN {X 0,Y 447.944,Z 420.322,A -85,B 0,C 180,E1 -8810.518,E2 -8810.518} C_VEL
LIN {X 0,Y 447.647,Z 429.863,A -85,B 0,C 180,E1 -8811.195,E2 -8811.195} C_VEL
LIN {X 0,Y 447.247,Z 439.25,A -85,B 0,C 180,E1 -8812.079,E2 -8812.079} C_VEL
LIN {X 0,Y 446.884,Z 446.758,A -85,B 0,C 180,E1 -8812.999,E2 -8812.999} C_VEL
LIN {X 0,Y 446.587,Z 453.812,A -85,B 0,C 180,E1 -8814.129,E2 -8814.129} C_VEL
LIN {X 0,Y 446.31,Z 458.189,A -85,B 0,C 180,E1 -8815.032,E2 -8815.032} C_VEL
LIN {X 0,Y 446.254,Z 461.622,A -85,B 0,C 180,E1 -8815.936,E2 -8815.936} C_VEL
LIN {X 0,Y 446.035,Z 464.263,A -85,B 0,C 180,E1 -8816.839,E2 -8816.839} C_VEL
LIN {X 0,Y 445.792,Z 465.314,A -85,B 0,C 180,E1 -8817.289,E2 -8817.289} C_VEL
LIN {X 0,Y 445.669,Z 466.842,A -85,B 0,C 180,E1 -8818.193,E2 -8818.193} C_VEL
LIN {X 0,Y 445.61,Z 467.683,A -85,B 0,C 180,E1 -8819.096,E2 -8819.096} C_VEL
LIN {X 0,Y 445.579,Z 467.857,A -85,B 0,C 180,E1 -8820,E2 -8820} C_VEL
LIN {X 0,Y 445.569,Z 467.365,A -85,B 0,C 180,E1 -8820.904,E2 -8820.904} C_VEL
LIN {X 0,Y 445.603,Z 466.2,A -85,B 0,C 180,E1 -8821.808,E2 -8821.808} C_VEL
LIN {X 0,Y 445.914,Z 463.114,A -85,B 0,C 180,E1 -8823.162,E2 -8823.162} C_VEL
LIN {X 0,Y 446.116,Z 458.283,A -85,B 0,C 180,E1 -8824.518,E2 -8824.518} C_VEL
LIN {X 0,Y 446.317,Z 452.688,A -85,B 0,C 180,E1 -8825.648,E2 -8825.648} C_VEL
LIN {X 0,Y 446.418,Z 445.442,A -85,B 0,C 180,E1 -8826.758,E2 -8826.758} C_VEL
LIN {X 0,Y 446.692,Z 437.958,A -85,B 0,C 180,E1 -8827.64,E2 -8827.64} C_VEL
LIN {X 0,Y 446.967,Z 428.774,A -85,B 0,C 180,E1 -8828.477,E2 -8828.477} C_VEL
LIN {X 0,Y 447.26,Z 418.811,A -85,B 0,C 180,E1 -8829.155,E2 -8829.155} C_VEL
LIN {X 0,Y 445.692,Z 407.928,A -85,B 0,C 180,E1 -8829.717,E2 -8829.717} C_VEL
LIN {X 0,Y 445.621,Z 407.258,A -85,B 0,C 180,E1 -8829.761,E2 -8829.761} C_VEL
LIN {X 0,Y 445.729,Z 400.924,A -85,B 0,C 180,E1 -8832.753,E2 -8832.753} C_VEL
LIN {X 0,Y 445.906,Z 394.244,A -85,B 0,C 180,E1 -8835.964,E2 -8835.964} C_VEL
LIN {X 0,Y 446.022,Z 387.354,A -85,B 0,C 180,E1 -8839.323,E2 -8839.323} C_VEL
LIN {X 0,Y 446.113,Z 381.525,A -85,B 0,C 180,E1 -8842.216,E2 -8842.216} C_VEL
LIN {X 0,Y 446.311,Z 375.627,A -85,B 0,C 180,E1 -8845.161,E2 -8845.161} C_VEL
LIN {X 0,Y 446.488,Z 369.678,A -85,B 0,C 180,E1 -8848.179,E2 -8848.179} C_VEL
LIN {X 0,Y 446.596,Z 364.932,A -85,B 0,C 180,E1 -8850.629,E2 -8850.629} C_VEL
LIN {X 0,Y 446.434,Z 364.876,A -85,B 0,C 180,E1 -8854.523,E2 -8854.523} C_VEL
LIN {X 0,Y 446.434,Z 364.876,A -85,B 0,C 180,E1 -8858.082,E2 -8858.082} C_VEL
LIN {X 0,Y 446.43,Z 364.877,A -85,B 0,C 180,E1 -8860.918,E2 -8860.918} C_VEL
LIN {X 0,Y 446.405,Z 364.876,A -85,B 0,C 180,E1 -8863.846,E2 -8863.846} C_VEL
LIN {X 0,Y 446.424,Z 364.879,A -85,B 0,C 180,E1 -8866.4,E2 -8866.4} C_VEL
LIN {X 0,Y 446.447,Z 364.874,A -85,B 0,C 180,E1 -8869.802,E2 -8869.802} C_VEL
LIN {X 0,Y 446.405,Z 364.878,A -85,B 0,C 180,E1 -8873.255,E2 -8873.255} C_VEL
LIN {X 0,Y 446.451,Z 364.875,A -85,B 0,C 180,E1 -8876.566,E2 -8876.566} C_VEL
LIN {X 0,Y 446.435,Z 364.877,A -85,B 0,C 180,E1 -8879.979,E2 -8879.979} C_VEL
LIN {X 0,Y 446.48,Z 364.872,A -85,B 0,C 180,E1 -8882.839,E2 -8882.839} C_VEL
LIN {X 0,Y 446.466,Z 364.87,A -85,B 0,C 180,E1 -8885.924,E2 -8885.924} C_VEL
LIN {X 0,Y 446.457,Z 364.872,A -85,B 0,C 180,E1 -8888.773,E2 -8888.773} C_VEL
LIN {X 0,Y 446.461,Z 364.873,A -85,B 0,C 180,E1 -8891.649,E2 -8891.649} C_VEL
LIN {X 0,Y 446.512,Z 364.869,A -85,B 0,C 180,E1 -8894.48,E2 -8894.48} C_VEL
LIN {X 0,Y 446.522,Z 364.867,A -85,B 0,C 180,E1 -8898.193,E2 -8898.193} C_VEL
LIN {X 0,Y 446.604,Z 364.855,A -85,B 0,C 180,E1 -8901.858,E2 -8901.858} C_VEL
LIN {X 0,Y 446.646,Z 364.85,A -85,B 0,C 180,E1 -8904.583,E2 -8904.583} C_VEL
LIN {X 0,Y 446.467,Z 364.871,A -85,B 0,C 180,E1 -8906.17,E2 -8906.17} C_VEL
LIN {X 0,Y 445.88,Z 364.948,A -85,B 0,C 180,E1 -8906.923,E2 -8906.923} C_VEL
LIN {X 0,Y 443.226,Z 365.283,A -85,B 0,C 180,E1 -8908.15,E2 -8908.15} C_VEL
LIN {X 0,Y 440.914,Z 365.569,A -85,B 0,C 180,E1 -8909.14,E2 -8909.14} C_VEL
LIN {X 0,Y 439.855,Z 365.697,A -85,B 0,C 180,E1 -8909.902,E2 -8909.902} C_VEL
LIN {X 0,Y 439.735,Z 365.71,A -85,B 0,C 180,E1 -8910.16,E2 -8910.16} C_VEL
LIN {X 0,Y 439.659,Z 365.72,A -85,B 0,C 180,E1 -8912.749,E2 -8912.749} C_VEL
LIN {X 0,Y 439.615,Z 365.725,A -85,B 0,C 180,E1 -8916.425,E2 -8916.425} C_VEL
LIN {X 0,Y 439.504,Z 365.736,A -85,B 0,C 180,E1 -8919.201,E2 -8919.201} C_VEL
LIN {X 0,Y 439.469,Z 365.743,A -85,B 0,C 180,E1 -8922.937,E2 -8922.937} C_VEL
LIN {X 0,Y 439.451,Z 365.746,A -85,B 0,C 180,E1 -8926.349,E2 -8926.349} C_VEL
LIN {X 0,Y 439.435,Z 365.75,A -85,B 0,C 180,E1 -8929.625,E2 -8929.625} C_VEL
LIN {X 0,Y 439.368,Z 365.755,A -85,B 0,C 180,E1 -8932.575,E2 -8932.575} C_VEL
LIN {X 0,Y 439.408,Z 365.751,A -85,B 0,C 180,E1 -8935.585,E2 -8935.585} C_VEL
LIN {X 0,Y 439.421,Z 365.748,A -85,B 0,C 180,E1 -8938.673,E2 -8938.673} C_VEL
LIN {X 0,Y 439.373,Z 365.753,A -85,B 0,C 180,E1 -8942.03,E2 -8942.03} C_VEL
LIN {X 0,Y 439.397,Z 365.752,A -85,B 0,C 180,E1 -8945.34,E2 -8945.34} C_VEL
LIN {X 0,Y 439.388,Z 365.753,A -85,B 0,C 180,E1 -8948.595,E2 -8948.595} C_VEL
LIN {X 0,Y 439.391,Z 365.755,A -85,B 0,C 180,E1 -8951.257,E2 -8951.257} C_VEL
LIN {X 0,Y 439.404,Z 365.752,A -85,B 0,C 180,E1 -8954.729,E2 -8954.729} C_VEL
LIN {X 0,Y 439.398,Z 365.753,A -85,B 0,C 180,E1 -8957.796,E2 -8957.796} C_VEL
LIN {X 0,Y 439.428,Z 365.747,A -85,B 0,C 180,E1 -8960.227,E2 -8960.227} C_VEL
LIN {X 0,Y 439.376,Z 365.753,A -85,B 0,C 180,E1 -8963.713,E2 -8963.713} C_VEL
LIN {X 0,Y 439.375,Z 365.755,A -85,B 0,C 180,E1 -8967.054,E2 -8967.054} C_VEL
LIN {X 0,Y 439.385,Z 365.754,A -85,B 0,C 180,E1 -8970.274,E2 -8970.274} C_VEL
LIN {X 0,Y 439.431,Z 365.747,A -85,B 0,C 180,E1 -8973.396,E2 -8973.396} C_VEL
LIN {X 0,Y 439.39,Z 365.754,A -85,B 0,C 180,E1 -8976.43,E2 -8976.43} C_VEL
LIN {X 0,Y 439.392,Z 365.754,A -85,B 0,C 180,E1 -8979.397,E2 -8979.397} C_VEL
LIN {X 0,Y 439.434,Z 365.747,A -85,B 0,C 180,E1 -8982.31,E2 -8982.31} C_VEL
LIN {X 0,Y 439.45,Z 365.744,A -85,B 0,C 180,E1 -8985.174,E2 -8985.174} C_VEL
LIN {X 0,Y 439.51,Z 365.738,A -85,B 0,C 180,E1 -8988.002,E2 -8988.002} C_VEL
LIN {X 0,Y 439.551,Z 365.733,A -85,B 0,C 180,E1 -8991.726,E2 -8991.726} C_VEL
LIN {X 0,Y 439.623,Z 365.725,A -85,B 0,C 180,E1 -8994.496,E2 -8994.496} C_VEL
LIN {X 0,Y 439.637,Z 365.724,A -85,B 0,C 180,E1 -8998.168,E2 -8998.168} C_VEL
LIN {X 0,Y 439.767,Z 365.707,A -85,B 0,C 180,E1 -9000,E2 -9000} C_VEL
LIN {X 0,Y 439.658,Z 365.721,A -85,B 0,C 180,E1 -9002.749,E2 -9002.749} C_VEL
LIN {X 0,Y 439.621,Z 365.728,A -85,B 0,C 180,E1 -9006.425,E2 -9006.425} C_VEL
LIN {X 0,Y 439.502,Z 365.738,A -85,B 0,C 180,E1 -9009.202,E2 -9009.202} C_VEL
LIN {X 0,Y 439.468,Z 365.744,A -85,B 0,C 180,E1 -9012.938,E2 -9012.938} C_VEL
LIN {X 0,Y 439.448,Z 365.749,A -85,B 0,C 180,E1 -9016.348,E2 -9016.348} C_VEL
LIN {X 0,Y 439.404,Z 365.751,A -85,B 0,C 180,E1 -9019.626,E2 -9019.626} C_VEL
LIN {X 0,Y 439.367,Z 365.756,A -85,B 0,C 180,E1 -9022.575,E2 -9022.575} C_VEL
LIN {X 0,Y 439.407,Z 365.75,A -85,B 0,C 180,E1 -9025.585,E2 -9025.585} C_VEL
LIN {X 0,Y 439.419,Z 365.747,A -85,B 0,C 180,E1 -9028.673,E2 -9028.673} C_VEL
LIN {X 0,Y 439.372,Z 365.756,A -85,B 0,C 180,E1 -9032.03,E2 -9032.03} C_VEL
LIN {X 0,Y 439.398,Z 365.753,A -85,B 0,C 180,E1 -9035.341,E2 -9035.341} C_VEL
LIN {X 0,Y 439.392,Z 365.751,A -85,B 0,C 180,E1 -9038.594,E2 -9038.594} C_VEL
LIN {X 0,Y 439.391,Z 365.752,A -85,B 0,C 180,E1 -9041.257,E2 -9041.257} C_VEL
LIN {X 0,Y 439.408,Z 365.75,A -85,B 0,C 180,E1 -9044.729,E2 -9044.729} C_VEL
LIN {X 0,Y 439.4,Z 365.753,A -85,B 0,C 180,E1 -9047.796,E2 -9047.796} C_VEL
LIN {X 0,Y 439.396,Z 365.75,A -85,B 0,C 180,E1 -9050.224,E2 -9050.224} C_VEL
LIN {X 0,Y 439.375,Z 365.756,A -85,B 0,C 180,E1 -9053.713,E2 -9053.713} C_VEL
LIN {X 0,Y 439.427,Z 365.772,A -85,B 0,C 180,E1 -9055.752,E2 -9055.752} C_VEL
LIN {X 0,Y 442.404,Z 379.654,A -85,B 0,C 180,E1 -9059.446,E2 -9059.446} C_VEL
LIN {X 0,Y 443.336,Z 384.504,A -85,B 0,C 180,E1 -9060.679,E2 -9060.679} C_VEL
LIN {X 0,Y 443.158,Z 389.417,A -85,B 0,C 180,E1 -9061.849,E2 -9061.849} C_VEL
LIN {X 0,Y 441.873,Z 404.36,A -85,B 0,C 180,E1 -9065.295,E2 -9065.295} C_VEL
LIN {X 0,Y 440.724,Z 420.706,A -85,B 0,C 180,E1 -9068.974,E2 -9068.974} C_VEL
LIN {X 0,Y 439.779,Z 438.059,A -85,B 0,C 180,E1 -9072.804,E2 -9072.804} C_VEL
LIN {X 0,Y 439.465,Z 444.586,A -85,B 0,C 180,E1 -9074.225,E2 -9074.225} C_VEL
LIN {X 0,Y 440.79,Z 457.806,A -85,B 0,C 180,E1 -9074.599,E2 -9074.599} C_VEL
LIN {X 0,Y 441.442,Z 466.617,A -85,B 0,C 180,E1 -9074.948,E2 -9074.948} C_VEL
LIN {X 0,Y 441.06,Z 479.118,A -85,B 0,C 180,E1 -9075.583,E2 -9075.583} C_VEL
LIN {X 0,Y 440.519,Z 491.288,A -85,B 0,C 180,E1 -9076.404,E2 -9076.404} C_VEL
LIN {X 0,Y 440.057,Z 502.985,A -85,B 0,C 180,E1 -9077.432,E2 -9077.432} C_VEL
LIN {X 0,Y 439.586,Z 510.527,A -85,B 0,C 180,E1 -9078.238,E2 -9078.238} C_VEL
LIN {X 0,Y 439.178,Z 519.519,A -85,B 0,C 180,E1 -9079.395,E2 -9079.395} C_VEL
LIN {X 0,Y 438.879,Z 526.905,A -85,B 0,C 180,E1 -9080.553,E2 -9080.553} C_VEL
LIN {X 0,Y 438.67,Z 534.122,A -85,B 0,C 180,E1 -9081.941,E2 -9081.941} C_VEL
LIN {X 0,Y 438.576,Z 538.969,A -85,B 0,C 180,E1 -9083.097,E2 -9083.097} C_VEL
LIN {X 0,Y 438.537,Z 543.613,A -85,B 0,C 180,E1 -9084.482,E2 -9084.482} C_VEL
LIN {X 0,Y 438.43,Z 546.02,A -85,B 0,C 180,E1 -9085.403,E2 -9085.403} C_VEL
LIN {X 0,Y 438.536,Z 547.99,A -85,B 0,C 180,E1 -9086.325,E2 -9086.325} C_VEL
LIN {X 0,Y 438.598,Z 549.515,A -85,B 0,C 180,E1 -9087.245,E2 -9087.245} C_VEL
LIN {X 0,Y 438.477,Z 550.541,A -85,B 0,C 180,E1 -9088.163,E2 -9088.163} C_VEL
LIN {X 0,Y 438.403,Z 551.375,A -85,B 0,C 180,E1 -9090,E2 -9090} C_VEL
LIN {X 0,Y 438.408,Z 551.145,A -85,B 0,C 180,E1 -9090.919,E2 -9090.919} C_VEL
LIN {X 0,Y 438.48,Z 550.489,A -85,B 0,C 180,E1 -9091.837,E2 -9091.837} C_VEL
LIN {X 0,Y 438.586,Z 549.429,A -85,B 0,C 180,E1 -9092.756,E2 -9092.756} C_VEL
LIN {X 0,Y 438.504,Z 546.975,A -85,B 0,C 180,E1 -9094.136,E2 -9094.136} C_VEL
LIN {X 0,Y 438.53,Z 543.483,A -85,B 0,C 180,E1 -9095.518,E2 -9095.518} C_VEL
LIN {X 0,Y 438.588,Z 538.053,A -85,B 0,C 180,E1 -9097.111,E2 -9097.111} C_VEL
LIN {X 0,Y 438.744,Z 531.807,A -85,B 0,C 180,E1 -9098.521,E2 -9098.521} C_VEL
LIN {X 0,Y 438.961,Z 524.139,A -85,B 0,C 180,E1 -9099.911,E2 -9099.911} C_VEL
LIN {X 0,Y 439.342,Z 516.317,A -85,B 0,C 180,E1 -9101.067,E2 -9101.067} C_VEL
LIN {X 0,Y 439.828,Z 506.741,A -85,B 0,C 180,E1 -9102.223,E2 -9102.223} C_VEL
LIN {X 0,Y 440.293,Z 497.132,A -85,B 0,C 180,E1 -9103.172,E2 -9103.172} C_VEL
LIN {X 0,Y 440.83,Z 485.894,A -85,B 0,C 180,E1 -9104.071,E2 -9104.071} C_VEL
LIN {X 0,Y 441.434,Z 473.785,A -85,B 0,C 180,E1 -9104.817,E2 -9104.817} C_VEL
LIN {X 0,Y 441.523,Z 463.733,A -85,B 0,C 180,E1 -9105.301,E2 -9105.301} C_VEL
LIN {X 0,Y 440.347,Z 449.694,A -85,B 0,C 180,E1 -9105.822,E2 -9105.822} C_VEL
LIN {X 0,Y 439.492,Z 443.556,A -85,B 0,C 180,E1 -9106.011,E2 -9106.011} C_VEL
LIN {X 0,Y 440.262,Z 428.422,A -85,B 0,C 180,E1 -9109.344,E2 -9109.344} C_VEL
LIN {X 0,Y 441.213,Z 414.802,A -85,B 0,C 180,E1 -9112.501,E2 -9112.501} C_VEL
LIN {X 0,Y 442.38,Z 402.959,A -85,B 0,C 180,E1 -9115.401,E2 -9115.401} C_VEL
LIN {X 0,Y 443.925,Z 391.832,A -85,B 0,C 180,E1 -9118.356,E2 -9118.356} C_VEL
LIN {X 0,Y 444.28,Z 387.789,A -85,B 0,C 180,E1 -9119.537,E2 -9119.537} C_VEL
LIN {X 0,Y 443.215,Z 381.925,A -85,B 0,C 180,E1 -9121.553,E2 -9121.553} C_VEL
LIN {X 0,Y 441.992,Z 376.223,A -85,B 0,C 180,E1 -9123.816,E2 -9123.816} C_VEL
LIN {X 0,Y 440.765,Z 371.385,A -85,B 0,C 180,E1 -9126.155,E2 -9126.155} C_VEL
LIN {X 0,Y 439.825,Z 367.494,A -85,B 0,C 180,E1 -9128.549,E2 -9128.549} C_VEL
LIN {X 0,Y 439.406,Z 365.753,A -85,B 0,C 180,E1 -9130.074,E2 -9130.074} C_VEL
LIN {X 0,Y 439.372,Z 365.757,A -85,B 0,C 180,E1 -9133.457,E2 -9133.457} C_VEL
LIN {X 0,Y 439.372,Z 365.756,A -85,B 0,C 180,E1 -9136.543,E2 -9136.543} C_VEL
LIN {X 0,Y 439.4,Z 365.754,A -85,B 0,C 180,E1 -9139.021,E2 -9139.021} C_VEL
LIN {X 0,Y 439.419,Z 365.752,A -85,B 0,C 180,E1 -9142.091,E2 -9142.091} C_VEL
LIN {X 0,Y 439.396,Z 365.844,A -85,B 0,C 180,E1 -9142.569,E2 -9142.569} C_VEL
LIN {X 0,Y 439.924,Z 368.212,A -85,B 0,C 180,E1 -9144.892,E2 -9144.892} C_VEL
LIN {X 0,Y 440.552,Z 371.718,A -85,B 0,C 180,E1 -9147.725,E2 -9147.725} C_VEL
LIN {X 0,Y 440.744,Z 374.142,A -85,B 0,C 180,E1 -9149.438,E2 -9149.438} C_VEL
LIN {X 0,Y 440.612,Z 377.199,A -85,B 0,C 180,E1 -9151.411,E2 -9151.411} C_VEL
LIN {X 0,Y 440.21,Z 382.197,A -85,B 0,C 180,E1 -9154.465,E2 -9154.465} C_VEL
LIN {X 0,Y 439.869,Z 388.229,A -85,B 0,C 180,E1 -9157.926,E2 -9157.926} C_VEL
LIN {X 0,Y 439.554,Z 394.436,A -85,B 0,C 180,E1 -9161.35,E2 -9161.35} C_VEL
LIN {X 0,Y 439.36,Z 399.773,A -85,B 0,C 180,E1 -9164.221,E2 -9164.221} C_VEL
LIN {X 0,Y 439.127,Z 406.991,A -85,B 0,C 180,E1 -9167.991,E2 -9167.991} C_VEL
LIN {X 0,Y 438.953,Z 410.129,A -85,B 0,C 180,E1 -9169.594,E2 -9169.594} C_VEL
LIN {X 0,Y 441.011,Z 420.57,A -85,B 0,C 180,E1 -9170.252,E2 -9170.252} C_VEL
LIN {X 0,Y 440.889,Z 428.67,A -85,B 0,C 180,E1 -9170.828,E2 -9170.828} C_VEL
LIN {X 0,Y 440.549,Z 437.333,A -85,B 0,C 180,E1 -9171.612,E2 -9171.612} C_VEL
LIN {X 0,Y 440.088,Z 445.23,A -85,B 0,C 180,E1 -9172.527,E2 -9172.527} C_VEL
LIN {X 0,Y 439.675,Z 452.245,A -85,B 0,C 180,E1 -9173.576,E2 -9173.576} C_VEL
LIN {X 0,Y 439.348,Z 458.131,A -85,B 0,C 180,E1 -9174.723,E2 -9174.723} C_VEL
LIN {X 0,Y 439.231,Z 462.498,A -85,B 0,C 180,E1 -9175.871,E2 -9175.871} C_VEL
LIN {X 0,Y 439.001,Z 465.094,A -85,B 0,C 180,E1 -9176.788,E2 -9176.788} C_VEL
LIN {X 0,Y 438.747,Z 466.125,A -85,B 0,C 180,E1 -9177.246,E2 -9177.246} C_VEL
LIN {X 0,Y 438.616,Z 467.615,A -85,B 0,C 180,E1 -9178.164,E2 -9178.164} C_VEL
LIN {X 0,Y 438.55,Z 468.42,A -85,B 0,C 180,E1 -9179.082,E2 -9179.082} C_VEL
LIN {X 0,Y 438.515,Z 468.557,A -85,B 0,C 180,E1 -9180,E2 -9180} C_VEL
LIN {X 0,Y 438.501,Z 468.025,A -85,B 0,C 180,E1 -9180.918,E2 -9180.918} C_VEL
LIN {X 0,Y 438.544,Z 466.816,A -85,B 0,C 180,E1 -9181.837,E2 -9181.837} C_VEL
LIN {X 0,Y 438.859,Z 463.668,A -85,B 0,C 180,E1 -9183.213,E2 -9183.213} C_VEL
LIN {X 0,Y 439.067,Z 458.779,A -85,B 0,C 180,E1 -9184.591,E2 -9184.591} C_VEL
LIN {X 0,Y 439.291,Z 453.132,A -85,B 0,C 180,E1 -9185.739,E2 -9185.739} C_VEL
LIN {X 0,Y 439.375,Z 446.059,A -85,B 0,C 180,E1 -9186.837,E2 -9186.837} C_VEL
LIN {X 0,Y 439.675,Z 438.319,A -85,B 0,C 180,E1 -9187.763,E2 -9187.763} C_VEL
LIN {X 0,Y 439.962,Z 429.114,A -85,B 0,C 180,E1 -9188.613,E2 -9188.613} C_VEL
LIN {X 0,Y 440.258,Z 419.155,A -85,B 0,C 180,E1 -9189.302,E2 -9189.302} C_VEL
LIN {X 0,Y 438.62,Z 408.222,A -85,B 0,C 180,E1 -9189.875,E2 -9189.875} C_VEL
LIN {X 0,Y 438.552,Z 407.527,A -85,B 0,C 180,E1 -9189.92,E2 -9189.92} C_VEL
LIN {X 0,Y 438.661,Z 401.161,A -85,B 0,C 180,E1 -9192.962,E2 -9192.962} C_VEL
LIN {X 0,Y 438.846,Z 394.729,A -85,B 0,C 180,E1 -9196.078,E2 -9196.078} C_VEL
LIN {X 0,Y 438.957,Z 387.489,A -85,B 0,C 180,E1 -9199.647,E2 -9199.647} C_VEL
LIN {X 0,Y 439.083,Z 381.6,A -85,B 0,C 180,E1 -9202.591,E2 -9202.591} C_VEL
LIN {X 0,Y 439.268,Z 375.663,A -85,B 0,C 180,E1 -9205.594,E2 -9205.594} C_VEL
LIN {X 0,Y 439.572,Z 368.678,A -85,B 0,C 180,E1 -9209.186,E2 -9209.186} C_VEL
LIN {X 0,Y 439.525,Z 365.739,A -85,B 0,C 180,E1 -9210.776,E2 -9210.776} C_VEL
LIN {X 0,Y 439.391,Z 365.751,A -85,B 0,C 180,E1 -9214.044,E2 -9214.044} C_VEL
LIN {X 0,Y 439.36,Z 365.757,A -85,B 0,C 180,E1 -9216.889,E2 -9216.889} C_VEL
LIN {X 0,Y 439.41,Z 365.75,A -85,B 0,C 180,E1 -9219.85,E2 -9219.85} C_VEL
LIN {X 0,Y 439.386,Z 365.754,A -85,B 0,C 180,E1 -9222.627,E2 -9222.627} C_VEL
LIN {X 0,Y 439.409,Z 365.749,A -85,B 0,C 180,E1 -9225.271,E2 -9225.271} C_VEL
LIN {X 0,Y 439.393,Z 365.753,A -85,B 0,C 180,E1 -9228.743,E2 -9228.743} C_VEL
LIN {X 0,Y 439.377,Z 365.754,A -85,B 0,C 180,E1 -9231.608,E2 -9231.608} C_VEL
LIN {X 0,Y 439.402,Z 365.752,A -85,B 0,C 180,E1 -9234.844,E2 -9234.844} C_VEL
LIN {X 0,Y 439.377,Z 365.757,A -85,B 0,C 180,E1 -9238.14,E2 -9238.14} C_VEL
LIN {X 0,Y 439.436,Z 365.747,A -85,B 0,C 180,E1 -9241.598,E2 -9241.598} C_VEL
LIN {X 0,Y 439.401,Z 365.753,A -85,B 0,C 180,E1 -9244.415,E2 -9244.415} C_VEL
LIN {X 0,Y 439.368,Z 365.754,A -85,B 0,C 180,E1 -9247.425,E2 -9247.425} C_VEL
LIN {X 0,Y 439.445,Z 365.746,A -85,B 0,C 180,E1 -9250.663,E2 -9250.663} C_VEL
LIN {X 0,Y 439.466,Z 365.744,A -85,B 0,C 180,E1 -9254.225,E2 -9254.225} C_VEL
LIN {X 0,Y 439.488,Z 365.743,A -85,B 0,C 180,E1 -9258.001,E2 -9258.001} C_VEL
LIN {X 0,Y 439.552,Z 365.734,A -85,B 0,C 180,E1 -9261.726,E2 -9261.726} C_VEL
LIN {X 0,Y 439.622,Z 365.726,A -85,B 0,C 180,E1 -9264.496,E2 -9264.496} C_VEL
LIN {X 0,Y 439.638,Z 365.724,A -85,B 0,C 180,E1 -9268.168,E2 -9268.168} C_VEL
LIN {X 0,Y 439.735,Z 365.71,A -85,B 0,C 180,E1 -9270.16,E2 -9270.16} C_VEL
LIN {X 0,Y 438.946,Z 365.808,A -85,B 0,C 180,E1 -9270.925,E2 -9270.925} C_VEL
LIN {X 0,Y 435.955,Z 366.181,A -85,B 0,C 180,E1 -9272.166,E2 -9272.166} C_VEL
LIN {X 0,Y 433.493,Z 366.487,A -85,B 0,C 180,E1 -9273.167,E2 -9273.167} C_VEL
LIN {X 0,Y 432.456,Z 366.617,A -85,B 0,C 180,E1 -9273.942,E2 -9273.942} C_VEL
LIN {X 0,Y 432.379,Z 366.625,A -85,B 0,C 180,E1 -9274.205,E2 -9274.205} C_VEL
LIN {X 0,Y 432.568,Z 366.602,A -85,B 0,C 180,E1 -9276.53,E2 -9276.53} C_VEL
LIN {X 0,Y 432.447,Z 366.617,A -85,B 0,C 180,E1 -9279.353,E2 -9279.353} C_VEL
LIN {X 0,Y 432.434,Z 366.619,A -85,B 0,C 180,E1 -9282.803,E2 -9282.803} C_VEL
LIN {X 0,Y 432.416,Z 366.621,A -85,B 0,C 180,E1 -9286.479,E2 -9286.479} C_VEL
LIN {X 0,Y 432.377,Z 366.627,A -85,B 0,C 180,E1 -9289.959,E2 -9289.959} C_VEL
LIN {X 0,Y 432.323,Z 366.633,A -85,B 0,C 180,E1 -9292.964,E2 -9292.964} C_VEL
LIN {X 0,Y 432.368,Z 366.629,A -85,B 0,C 180,E1 -9296.032,E2 -9296.032} C_VEL
LIN {X 0,Y 432.346,Z 366.63,A -85,B 0,C 180,E1 -9299.187,E2 -9299.187} C_VEL
LIN {X 0,Y 432.326,Z 366.631,A -85,B 0,C 180,E1 -9302.443,E2 -9302.443} C_VEL
LIN {X 0,Y 432.347,Z 366.631,A -85,B 0,C 180,E1 -9305.632,E2 -9305.632} C_VEL
LIN {X 0,Y 432.357,Z 366.63,A -85,B 0,C 180,E1 -9309.342,E2 -9309.342} C_VEL
LIN {X 0,Y 432.336,Z 366.63,A -85,B 0,C 180,E1 -9311.797,E2 -9311.797} C_VEL
LIN {X 0,Y 432.336,Z 366.63,A -85,B 0,C 180,E1 -9314.347,E2 -9314.347} C_VEL
LIN {X 0,Y 432.323,Z 366.634,A -85,B 0,C 180,E1 -9317.016,E2 -9317.016} C_VEL
LIN {X 0,Y 432.335,Z 366.631,A -85,B 0,C 180,E1 -9319.821,E2 -9319.821} C_VEL
LIN {X 0,Y 432.309,Z 366.637,A -85,B 0,C 180,E1 -9323.022,E2 -9323.022} C_VEL
LIN {X 0,Y 432.361,Z 366.628,A -85,B 0,C 180,E1 -9325.996,E2 -9325.996} C_VEL
LIN {X 0,Y 432.35,Z 366.631,A -85,B 0,C 180,E1 -9329.489,E2 -9329.489} C_VEL
LIN {X 0,Y 432.394,Z 366.627,A -85,B 0,C 180,E1 -9332.928,E2 -9332.928} C_VEL
LIN {X 0,Y 432.374,Z 366.625,A -85,B 0,C 180,E1 -9336.023,E2 -9336.023} C_VEL
LIN {X 0,Y 432.353,Z 366.63,A -85,B 0,C 180,E1 -9339.046,E2 -9339.046} C_VEL
LIN {X 0,Y 432.381,Z 366.625,A -85,B 0,C 180,E1 -9342.011,E2 -9342.011} C_VEL
LIN {X 0,Y 432.398,Z 366.625,A -85,B 0,C 180,E1 -9344.926,E2 -9344.926} C_VEL
LIN {X 0,Y 432.483,Z 366.612,A -85,B 0,C 180,E1 -9347.804,E2 -9347.804} C_VEL
LIN {X 0,Y 432.495,Z 366.611,A -85,B 0,C 180,E1 -9351.59,E2 -9351.59} C_VEL
LIN {X 0,Y 432.6,Z 366.599,A -85,B 0,C 180,E1 -9354.406,E2 -9354.406} C_VEL
LIN {X 0,Y 432.607,Z 366.599,A -85,B 0,C 180,E1 -9358.138,E2 -9358.138} C_VEL
LIN {X 0,Y 432.737,Z 366.583,A -85,B 0,C 180,E1 -9360,E2 -9360} C_VEL
LIN {X 0,Y 432.608,Z 366.6,A -85,B 0,C 180,E1 -9362.793,E2 -9362.793} C_VEL
LIN {X 0,Y 432.575,Z 366.604,A -85,B 0,C 180,E1 -9366.53,E2 -9366.53} C_VEL
LIN {X 0,Y 432.445,Z 366.617,A -85,B 0,C 180,E1 -9369.353,E2 -9369.353} C_VEL
LIN {X 0,Y 432.433,Z 366.621,A -85,B 0,C 180,E1 -9372.803,E2 -9372.803} C_VEL
LIN {X 0,Y 432.414,Z 366.624,A -85,B 0,C 180,E1 -9376.479,E2 -9376.479} C_VEL
LIN {X 0,Y 432.341,Z 366.634,A -85,B 0,C 180,E1 -9379.96,E2 -9379.96} C_VEL
LIN {X 0,Y 432.321,Z 366.633,A -85,B 0,C 180,E1 -9382.964,E2 -9382.964} C_VEL
LIN {X 0,Y 432.366,Z 366.629,A -85,B 0,C 180,E1 -9386.032,E2 -9386.032} C_VEL
LIN {X 0,Y 432.345,Z 366.628,A -85,B 0,C 180,E1 -9389.187,E2 -9389.187} C_VEL
LIN {X 0,Y 432.325,Z 366.633,A -85,B 0,C 180,E1 -9392.443,E2 -9392.443} C_VEL
LIN {X 0,Y 432.347,Z 366.63,A -85,B 0,C 180,E1 -9395.632,E2 -9395.632} C_VEL
LIN {X 0,Y 432.354,Z 366.627,A -85,B 0,C 180,E1 -9398.717,E2 -9398.717} C_VEL
LIN {X 0,Y 432.337,Z 366.633,A -85,B 0,C 180,E1 -9401.797,E2 -9401.797} C_VEL
LIN {X 0,Y 432.343,Z 366.632,A -85,B 0,C 180,E1 -9404.346,E2 -9404.346} C_VEL
LIN {X 0,Y 432.327,Z 366.633,A -85,B 0,C 180,E1 -9407.015,E2 -9407.015} C_VEL
LIN {X 0,Y 432.335,Z 366.634,A -85,B 0,C 180,E1 -9409.821,E2 -9409.821} C_VEL
LIN {X 0,Y 432.308,Z 366.637,A -85,B 0,C 180,E1 -9413.022,E2 -9413.022} C_VEL
LIN {X 0,Y 432.416,Z 366.808,A -85,B 0,C 180,E1 -9415.474,E2 -9415.474} C_VEL
LIN {X 0,Y 435.348,Z 380.392,A -85,B 0,C 180,E1 -9419.166,E2 -9419.166} C_VEL
LIN {X 0,Y 436.446,Z 386.613,A -85,B 0,C 180,E1 -9420.783,E2 -9420.783} C_VEL
LIN {X 0,Y 435.751,Z 395.121,A -85,B 0,C 180,E1 -9422.812,E2 -9422.812} C_VEL
LIN {X 0,Y 434.469,Z 410.512,A -85,B 0,C 180,E1 -9426.399,E2 -9426.399} C_VEL
LIN {X 0,Y 433.332,Z 427.022,A -85,B 0,C 180,E1 -9430.165,E2 -9430.165} C_VEL
LIN {X 0,Y 432.528,Z 441.754,A -85,B 0,C 180,E1 -9433.47,E2 -9433.47} C_VEL
LIN {X 0,Y 432.441,Z 444.232,A -85,B 0,C 180,E1 -9434.022,E2 -9434.022} C_VEL
LIN {X 0,Y 433.891,Z 459.591,A -85,B 0,C 180,E1 -9434.499,E2 -9434.499} C_VEL
LIN {X 0,Y 434.427,Z 467.115,A -85,B 0,C 180,E1 -9434.819,E2 -9434.819} C_VEL
LIN {X 0,Y 434.033,Z 479.38,A -85,B 0,C 180,E1 -9435.464,E2 -9435.464} C_VEL
LIN {X 0,Y 433.497,Z 491.179,A -85,B 0,C 180,E1 -9436.285,E2 -9436.285} C_VEL
LIN {X 0,Y 433.001,Z 502.931,A -85,B 0,C 180,E1 -9437.343,E2 -9437.343} C_VEL
LIN {X 0,Y 432.498,Z 511.377,A -85,B 0,C 180,E1 -9438.28,E2 -9438.28} C_VEL
LIN {X 0,Y 432.055,Z 520.13,A -85,B 0,C 180,E1 -9439.456,E2 -9439.456} C_VEL
LIN {X 0,Y 431.729,Z 528.564,A -85,B 0,C 180,E1 -9440.868,E2 -9440.868} C_VEL
LIN {X 0,Y 431.55,Z 535.307,A -85,B 0,C 180,E1 -9442.279,E2 -9442.279} C_VEL
LIN {X 0,Y 431.423,Z 540.227,A -85,B 0,C 180,E1 -9443.57,E2 -9443.57} C_VEL
LIN {X 0,Y 431.404,Z 544.098,A -85,B 0,C 180,E1 -9444.859,E2 -9444.859} C_VEL
LIN {X 0,Y 431.469,Z 547.253,A -85,B 0,C 180,E1 -9446.264,E2 -9446.264} C_VEL
LIN {X 0,Y 431.546,Z 548.798,A -85,B 0,C 180,E1 -9447.2,E2 -9447.2} C_VEL
LIN {X 0,Y 431.424,Z 549.841,A -85,B 0,C 180,E1 -9448.133,E2 -9448.133} C_VEL
LIN {X 0,Y 431.345,Z 550.466,A -85,B 0,C 180,E1 -9449.066,E2 -9449.066} C_VEL
LIN {X 0,Y 431.339,Z 550.691,A -85,B 0,C 180,E1 -9450,E2 -9450} C_VEL
LIN {X 0,Y 431.348,Z 550.477,A -85,B 0,C 180,E1 -9450.934,E2 -9450.934} C_VEL
LIN {X 0,Y 431.426,Z 549.828,A -85,B 0,C 180,E1 -9451.867,E2 -9451.867} C_VEL
LIN {X 0,Y 431.504,Z 548.768,A -85,B 0,C 180,E1 -9452.801,E2 -9452.801} C_VEL
LIN {X 0,Y 431.405,Z 546.318,A -85,B 0,C 180,E1 -9454.204,E2 -9454.204} C_VEL
LIN {X 0,Y 431.452,Z 542.835,A -85,B 0,C 180,E1 -9455.609,E2 -9455.609} C_VEL
LIN {X 0,Y 431.512,Z 538.217,A -85,B 0,C 180,E1 -9457.016,E2 -9457.016} C_VEL
LIN {X 0,Y 431.681,Z 531.185,A -85,B 0,C 180,E1 -9458.662,E2 -9458.662} C_VEL
LIN {X 0,Y 431.897,Z 523.517,A -85,B 0,C 180,E1 -9460.075,E2 -9460.075} C_VEL
LIN {X 0,Y 432.321,Z 515.716,A -85,B 0,C 180,E1 -9461.249,E2 -9461.249} C_VEL
LIN {X 0,Y 432.845,Z 506.195,A -85,B 0,C 180,E1 -9462.421,E2 -9462.421} C_VEL
LIN {X 0,Y 433.355,Z 496.225,A -85,B 0,C 180,E1 -9463.421,E2 -9463.421} C_VEL
LIN {X 0,Y 433.916,Z 485.394,A -85,B 0,C 180,E1 -9464.3,E2 -9464.3} C_VEL
LIN {X 0,Y 434.566,Z 473.373,A -85,B 0,C 180,E1 -9465.057,E2 -9465.057} C_VEL
LIN {X 0,Y 434.691,Z 465.147,A -85,B 0,C 180,E1 -9465.472,E2 -9465.472} C_VEL
LIN {X 0,Y 433.698,Z 452.409,A -85,B 0,C 180,E1 -9465.991,E2 -9465.991} C_VEL
LIN {X 0,Y 432.501,Z 443.235,A -85,B 0,C 180,E1 -9466.288,E2 -9466.288} C_VEL
LIN {X 0,Y 433.415,Z 427.258,A -85,B 0,C 180,E1 -9469.909,E2 -9469.909} C_VEL
LIN {X 0,Y 434.323,Z 414.926,A -85,B 0,C 180,E1 -9472.852,E2 -9472.852} C_VEL
LIN {X 0,Y 435.631,Z 403.25,A -85,B 0,C 180,E1 -9475.823,E2 -9475.823} C_VEL
LIN {X 0,Y 437.292,Z 392.327,A -85,B 0,C 180,E1 -9478.826,E2 -9478.826} C_VEL
LIN {X 0,Y 437.399,Z 388.941,A -85,B 0,C 180,E1 -9479.874,E2 -9479.874} C_VEL
LIN {X 0,Y 435.987,Z 381.643,A -85,B 0,C 180,E1 -9482.56,E2 -9482.56} C_VEL
LIN {X 0,Y 434.708,Z 376.098,A -85,B 0,C 180,E1 -9485.025,E2 -9485.025} C_VEL
LIN {X 0,Y 433.342,Z 370.84,A -85,B 0,C 180,E1 -9488.046,E2 -9488.046} C_VEL
LIN {X 0,Y 432.619,Z 367.807,A -85,B 0,C 180,E1 -9490.527,E2 -9490.527} C_VEL
LIN {X 0,Y 432.361,Z 366.631,A -85,B 0,C 180,E1 -9492.089,E2 -9492.089} C_VEL
LIN {X 0,Y 432.344,Z 366.632,A -85,B 0,C 180,E1 -9495.664,E2 -9495.664} C_VEL
LIN {X 0,Y 432.37,Z 366.629,A -85,B 0,C 180,E1 -9498.393,E2 -9498.393} C_VEL
LIN {X 0,Y 432.378,Z 366.767,A -85,B 0,C 180,E1 -9500.924,E2 -9500.924} C_VEL
LIN {X 0,Y 432.977,Z 369.593,A -85,B 0,C 180,E1 -9504.252,E2 -9504.252} C_VEL
LIN {X 0,Y 433.641,Z 373.228,A -85,B 0,C 180,E1 -9507.433,E2 -9507.433} C_VEL
LIN {X 0,Y 433.851,Z 376.534,A -85,B 0,C 180,E1 -9509.856,E2 -9509.856} C_VEL
LIN {X 0,Y 433.49,Z 381.377,A -85,B 0,C 180,E1 -9513.002,E2 -9513.002} C_VEL
LIN {X 0,Y 433.094,Z 386.429,A -85,B 0,C 180,E1 -9516.066,E2 -9516.066} C_VEL
LIN {X 0,Y 432.776,Z 391.629,A -85,B 0,C 180,E1 -9519.068,E2 -9519.068} C_VEL
LIN {X 0,Y 432.502,Z 396.931,A -85,B 0,C 180,E1 -9522.017,E2 -9522.017} C_VEL
LIN {X 0,Y 432.261,Z 402.281,A -85,B 0,C 180,E1 -9524.922,E2 -9524.922} C_VEL
LIN {X 0,Y 432.135,Z 407.69,A -85,B 0,C 180,E1 -9527.794,E2 -9527.794} C_VEL
LIN {X 0,Y 431.958,Z 410.613,A -85,B 0,C 180,E1 -9529.305,E2 -9529.305} C_VEL
LIN {X 0,Y 434.28,Z 422.558,A -85,B 0,C 180,E1 -9530.099,E2 -9530.099} C_VEL
LIN {X 0,Y 433.927,Z 431.721,A -85,B 0,C 180,E1 -9530.797,E2 -9530.797} C_VEL
LIN {X 0,Y 433.526,Z 439.991,A -85,B 0,C 180,E1 -9531.611,E2 -9531.611} C_VEL
LIN {X 0,Y 433.093,Z 447.433,A -85,B 0,C 180,E1 -9532.541,E2 -9532.541} C_VEL
LIN {X 0,Y 432.657,Z 454.644,A -85,B 0,C 180,E1 -9533.705,E2 -9533.705} C_VEL
LIN {X 0,Y 432.292,Z 460.084,A -85,B 0,C 180,E1 -9534.87,E2 -9534.87} C_VEL
LIN {X 0,Y 432.209,Z 463.396,A -85,B 0,C 180,E1 -9535.804,E2 -9535.804} C_VEL
LIN {X 0,Y 431.968,Z 465.929,A -85,B 0,C 180,E1 -9536.736,E2 -9536.736} C_VEL
LIN {X 0,Y 431.703,Z 466.936,A -85,B 0,C 180,E1 -9537.201,E2 -9537.201} C_VEL
LIN {X 0,Y 431.562,Z 468.384,A -85,B 0,C 180,E1 -9538.134,E2 -9538.134} C_VEL
LIN {X 0,Y 431.489,Z 469.152,A -85,B 0,C 180,E1 -9539.067,E2 -9539.067} C_VEL
LIN {X 0,Y 431.45,Z 469.252,A -85,B 0,C 180,E1 -9540,E2 -9540} C_VEL
LIN {X 0,Y 431.435,Z 468.68,A -85,B 0,C 180,E1 -9540.933,E2 -9540.933} C_VEL
LIN {X 0,Y 431.488,Z 467.428,A -85,B 0,C 180,E1 -9541.867,E2 -9541.867} C_VEL
LIN {X 0,Y 431.807,Z 464.211,A -85,B 0,C 180,E1 -9543.266,E2 -9543.266} C_VEL
LIN {X 0,Y 431.993,Z 461.112,A -85,B 0,C 180,E1 -9544.198,E2 -9544.198} C_VEL
LIN {X 0,Y 432.129,Z 456.017,A -85,B 0,C 180,E1 -9545.366,E2 -9545.366} C_VEL
LIN {X 0,Y 432.301,Z 449.258,A -85,B 0,C 180,E1 -9546.535,E2 -9546.535} C_VEL
LIN {X 0,Y 432.469,Z 442.301,A -85,B 0,C 180,E1 -9547.47,E2 -9547.47} C_VEL
LIN {X 0,Y 432.799,Z 433.347,A -85,B 0,C 180,E1 -9548.404,E2 -9548.404} C_VEL
LIN {X 0,Y 433.146,Z 424.619,A -85,B 0,C 180,E1 -9549.102,E2 -9549.102} C_VEL
LIN {X 0,Y 433.042,Z 418.189,A -85,B 0,C 180,E1 -9549.517,E2 -9549.517} C_VEL
LIN {X 0,Y 431.465,Z 407.787,A -85,B 0,C 180,E1 -9550.085,E2 -9550.085} C_VEL
LIN {X 0,Y 431.634,Z 403.116,A -85,B 0,C 180,E1 -9552.328,E2 -9552.328} C_VEL
LIN {X 0,Y 431.787,Z 395.201,A -85,B 0,C 180,E1 -9556.195,E2 -9556.195} C_VEL
LIN {X 0,Y 431.926,Z 387.601,A -85,B 0,C 180,E1 -9559.98,E2 -9559.98} C_VEL
LIN {X 0,Y 432.046,Z 381.681,A -85,B 0,C 180,E1 -9562.98,E2 -9562.98} C_VEL
LIN {X 0,Y 432.249,Z 375.698,A -85,B 0,C 180,E1 -9566.04,E2 -9566.04} C_VEL
LIN {X 0,Y 432.568,Z 368.629,A -85,B 0,C 180,E1 -9569.705,E2 -9569.705} C_VEL
LIN {X 0,Y 432.461,Z 366.619,A -85,B 0,C 180,E1 -9570.907,E2 -9570.907} C_VEL
LIN {X 0,Y 432.344,Z 366.633,A -85,B 0,C 180,E1 -9574.677,E2 -9574.677} C_VEL
LIN {X 0,Y 432.35,Z 366.63,A -85,B 0,C 180,E1 -9578.149,E2 -9578.149} C_VEL
LIN {X 0,Y 432.336,Z 366.63,A -85,B 0,C 180,E1 -9581.602,E2 -9581.602} C_VEL
LIN {X 0,Y 432.337,Z 366.631,A -85,B 0,C 180,E1 -9584.347,E2 -9584.347} C_VEL
LIN {X 0,Y 432.328,Z 366.632,A -85,B 0,C 180,E1 -9587.015,E2 -9587.015} C_VEL
LIN {X 0,Y 432.336,Z 366.631,A -85,B 0,C 180,E1 -9589.821,E2 -9589.821} C_VEL
LIN {X 0,Y 432.31,Z 366.635,A -85,B 0,C 180,E1 -9593.022,E2 -9593.022} C_VEL
LIN {X 0,Y 432.362,Z 366.627,A -85,B 0,C 180,E1 -9595.997,E2 -9595.997} C_VEL
LIN {X 0,Y 432.351,Z 366.629,A -85,B 0,C 180,E1 -9599.49,E2 -9599.49} C_VEL
LIN {X 0,Y 432.395,Z 366.625,A -85,B 0,C 180,E1 -9602.928,E2 -9602.928} C_VEL
LIN {X 0,Y 432.372,Z 366.627,A -85,B 0,C 180,E1 -9606.023,E2 -9606.023} C_VEL
LIN {X 0,Y 432.354,Z 366.629,A -85,B 0,C 180,E1 -9609.046,E2 -9609.046} C_VEL
LIN {X 0,Y 432.381,Z 366.626,A -85,B 0,C 180,E1 -9612.011,E2 -9612.011} C_VEL
LIN {X 0,Y 432.399,Z 366.623,A -85,B 0,C 180,E1 -9614.926,E2 -9614.926} C_VEL
LIN {X 0,Y 432.463,Z 366.616,A -85,B 0,C 180,E1 -9617.803,E2 -9617.803} C_VEL
LIN {X 0,Y 432.496,Z 366.613,A -85,B 0,C 180,E1 -9621.59,E2 -9621.59} C_VEL
LIN {X 0,Y 432.598,Z 366.602,A -85,B 0,C 180,E1 -9624.406,E2 -9624.406} C_VEL
LIN {X 0,Y 432.608,Z 366.6,A -85,B 0,C 180,E1 -9628.138,E2 -9628.138} C_VEL
LIN {X 0,Y 432.707,Z 366.586,A -85,B 0,C 180,E1 -9630.135,E2 -9630.135} C_VEL
LIN {X 0,Y 432.608,Z 366.598,A -85,B 0,C 180,E1 -9632.793,E2 -9632.793} C_VEL
LIN {X 0,Y 432.379,Z 366.625,A -85,B 0,C 180,E1 -9634.205,E2 -9634.205} C_VEL
LIN {X 0,Y 431.747,Z 366.705,A -85,B 0,C 180,E1 -9634.983,E2 -9634.983} C_VEL
LIN {X 0,Y 428.962,Z 367.053,A -85,B 0,C 180,E1 -9636.25,E2 -9636.25} C_VEL
LIN {X 0,Y 426.583,Z 367.348,A -85,B 0,C 180,E1 -9637.272,E2 -9637.272} C_VEL
LIN {X 0,Y 425.546,Z 367.479,A -85,B 0,C 180,E1 -9638.06,E2 -9638.06} C_VEL
LIN {X 0,Y 425.454,Z 367.486,A -85,B 0,C 180,E1 -9638.328,E2 -9638.328} C_VEL
LIN {X 0,Y 425.356,Z 367.502,A -85,B 0,C 180,E1 -9641.436,E2 -9641.436} C_VEL
LIN {X 0,Y 425.352,Z 367.502,A -85,B 0,C 180,E1 -9644.35,E2 -9644.35} C_VEL
LIN {X 0,Y 425.346,Z 367.502,A -85,B 0,C 180,E1 -9647.302,E2 -9647.302} C_VEL
LIN {X 0,Y 425.317,Z 367.504,A -85,B 0,C 180,E1 -9650.304,E2 -9650.304} C_VEL
LIN {X 0,Y 425.31,Z 367.509,A -85,B 0,C 180,E1 -9653.365,E2 -9653.365} C_VEL
LIN {X 0,Y 425.351,Z 367.502,A -85,B 0,C 180,E1 -9656.844,E2 -9656.844} C_VEL
LIN {X 0,Y 425.294,Z 367.51,A -85,B 0,C 180,E1 -9659.719,E2 -9659.719} C_VEL
LIN {X 0,Y 425.285,Z 367.511,A -85,B 0,C 180,E1 -9663.048,E2 -9663.048} C_VEL
LIN {X 0,Y 425.285,Z 367.511,A -85,B 0,C 180,E1 -9665.929,E2 -9665.929} C_VEL
LIN {X 0,Y 425.303,Z 367.507,A -85,B 0,C 180,E1 -9669.044,E2 -9669.044} C_VEL
LIN {X 0,Y 425.277,Z 367.509,A -85,B 0,C 180,E1 -9672.653,E2 -9672.653} C_VEL
LIN {X 0,Y 425.264,Z 367.512,A -85,B 0,C 180,E1 -9676.044,E2 -9676.044} C_VEL
LIN {X 0,Y 425.276,Z 367.512,A -85,B 0,C 180,E1 -9678.621,E2 -9678.621} C_VEL
LIN {X 0,Y 425.308,Z 367.508,A -85,B 0,C 180,E1 -9681.102,E2 -9681.102} C_VEL
LIN {X 0,Y 425.302,Z 367.508,A -85,B 0,C 180,E1 -9684.664,E2 -9684.664} C_VEL
LIN {X 0,Y 425.267,Z 367.512,A -85,B 0,C 180,E1 -9688.073,E2 -9688.073} C_VEL
LIN {X 0,Y 425.334,Z 367.505,A -85,B 0,C 180,E1 -9691.368,E2 -9691.368} C_VEL
LIN {X 0,Y 425.298,Z 367.508,A -85,B 0,C 180,E1 -9694.555,E2 -9694.555} C_VEL
LIN {X 0,Y 425.29,Z 367.509,A -85,B 0,C 180,E1 -9697.661,E2 -9697.661} C_VEL
LIN {X 0,Y 425.365,Z 367.5,A -85,B 0,C 180,E1 -9700.704,E2 -9700.704} C_VEL
LIN {X 0,Y 425.391,Z 367.494,A -85,B 0,C 180,E1 -9703.688,E2 -9703.688} C_VEL
LIN {X 0,Y 425.433,Z 367.49,A -85,B 0,C 180,E1 -9707.599,E2 -9707.599} C_VEL
LIN {X 0,Y 425.445,Z 367.489,A -85,B 0,C 180,E1 -9711.45,E2 -9711.45} C_VEL
LIN {X 0,Y 425.557,Z 367.476,A -85,B 0,C 180,E1 -9714.313,E2 -9714.313} C_VEL
LIN {X 0,Y 425.576,Z 367.474,A -85,B 0,C 180,E1 -9718.107,E2 -9718.107} C_VEL
LIN {X 0,Y 425.706,Z 367.459,A -85,B 0,C 180,E1 -9720,E2 -9720} C_VEL
LIN {X 0,Y 425.559,Z 367.478,A -85,B 0,C 180,E1 -9722.84,E2 -9722.84} C_VEL
LIN {X 0,Y 425.534,Z 367.48,A -85,B 0,C 180,E1 -9726.639,E2 -9726.639} C_VEL
LIN {X 0,Y 425.403,Z 367.494,A -85,B 0,C 180,E1 -9729.509,E2 -9729.509} C_VEL
LIN {X 0,Y 425.396,Z 367.497,A -85,B 0,C 180,E1 -9732.904,E2 -9732.904} C_VEL
LIN {X 0,Y 425.363,Z 367.5,A -85,B 0,C 180,E1 -9736.605,E2 -9736.605} C_VEL
LIN {X 0,Y 425.33,Z 367.504,A -85,B 0,C 180,E1 -9739.636,E2 -9739.636} C_VEL
LIN {X 0,Y 425.309,Z 367.507,A -85,B 0,C 180,E1 -9743.365,E2 -9743.365} C_VEL
LIN {X 0,Y 425.349,Z 367.5,A -85,B 0,C 180,E1 -9746.844,E2 -9746.844} C_VEL
LIN {X 0,Y 425.293,Z 367.51,A -85,B 0,C 180,E1 -9749.719,E2 -9749.719} C_VEL
LIN {X 0,Y 425.284,Z 367.509,A -85,B 0,C 180,E1 -9753.048,E2 -9753.048} C_VEL
LIN {X 0,Y 425.287,Z 367.51,A -85,B 0,C 180,E1 -9755.929,E2 -9755.929} C_VEL
LIN {X 0,Y 425.305,Z 367.505,A -85,B 0,C 180,E1 -9759.044,E2 -9759.044} C_VEL
LIN {X 0,Y 425.294,Z 367.509,A -85,B 0,C 180,E1 -9761.959,E2 -9761.959} C_VEL
LIN {X 0,Y 425.293,Z 367.511,A -85,B 0,C 180,E1 -9765.282,E2 -9765.282} C_VEL
LIN {X 0,Y 425.277,Z 367.509,A -85,B 0,C 180,E1 -9768.622,E2 -9768.622} C_VEL
LIN {X 0,Y 425.299,Z 367.505,A -85,B 0,C 180,E1 -9771.101,E2 -9771.101} C_VEL
LIN {X 0,Y 425.309,Z 367.509,A -85,B 0,C 180,E1 -9774.665,E2 -9774.665} C_VEL
LIN {X 0,Y 425.347,Z 367.649,A -85,B 0,C 180,E1 -9775.138,E2 -9775.138} C_VEL
LIN {X 0,Y 428.054,Z 380.157,A -85,B 0,C 180,E1 -9778.623,E2 -9778.623} C_VEL
LIN {X 0,Y 429.474,Z 387.608,A -85,B 0,C 180,E1 -9780.598,E2 -9780.598} C_VEL
LIN {X 0,Y 429.13,Z 393.274,A -85,B 0,C 180,E1 -9781.993,E2 -9781.993} C_VEL
LIN {X 0,Y 427.742,Z 407.906,A -85,B 0,C 180,E1 -9785.489,E2 -9785.489} C_VEL
LIN {X 0,Y 426.562,Z 422.899,A -85,B 0,C 180,E1 -9789.001,E2 -9789.001} C_VEL
LIN {X 0,Y 425.694,Z 437.94,A -85,B 0,C 180,E1 -9792.464,E2 -9792.464} C_VEL
LIN {X 0,Y 425.399,Z 443.982,A -85,B 0,C 180,E1 -9793.843,E2 -9793.843} C_VEL
LIN {X 0,Y 426.875,Z 459.336,A -85,B 0,C 180,E1 -9794.329,E2 -9794.329} C_VEL
LIN {X 0,Y 427.426,Z 468.759,A -85,B 0,C 180,E1 -9794.747,E2 -9794.747} C_VEL
LIN {X 0,Y 427.01,Z 479.541,A -85,B 0,C 180,E1 -9795.342,E2 -9795.342} C_VEL
LIN {X 0,Y 426.531,Z 490.148,A -85,B 0,C 180,E1 -9796.092,E2 -9796.092} C_VEL
LIN {X 0,Y 425.987,Z 501.99,A -85,B 0,C 180,E1 -9797.166,E2 -9797.166} C_VEL
LIN {X 0,Y 425.413,Z 510.205,A -85,B 0,C 180,E1 -9798.082,E2 -9798.082} C_VEL
LIN {X 0,Y 425.027,Z 519.074,A -85,B 0,C 180,E1 -9799.279,E2 -9799.279} C_VEL
LIN {X 0,Y 424.724,Z 526.348,A -85,B 0,C 180,E1 -9800.475,E2 -9800.475} C_VEL
LIN {X 0,Y 424.505,Z 533.406,A -85,B 0,C 180,E1 -9801.91,E2 -9801.91} C_VEL
LIN {X 0,Y 424.353,Z 539.754,A -85,B 0,C 180,E1 -9803.567,E2 -9803.567} C_VEL
LIN {X 0,Y 424.346,Z 543.314,A -85,B 0,C 180,E1 -9804.774,E2 -9804.774} C_VEL
LIN {X 0,Y 424.404,Z 546.504,A -85,B 0,C 180,E1 -9806.202,E2 -9806.202} C_VEL
LIN {X 0,Y 424.477,Z 548.064,A -85,B 0,C 180,E1 -9807.153,E2 -9807.153} C_VEL
LIN {X 0,Y 424.372,Z 549.135,A -85,B 0,C 180,E1 -9808.102,E2 -9808.102} C_VEL
LIN {X 0,Y 424.286,Z 549.769,A -85,B 0,C 180,E1 -9809.051,E2 -9809.051} C_VEL
LIN {X 0,Y 424.277,Z 550.003,A -85,B 0,C 180,E1 -9810,E2 -9810} C_VEL
LIN {X 0,Y 424.289,Z 549.81,A -85,B 0,C 180,E1 -9810.949,E2 -9810.949} C_VEL
LIN {X 0,Y 424.373,Z 549.167,A -85,B 0,C 180,E1 -9811.898,E2 -9811.898} C_VEL
LIN {X 0,Y 424.427,Z 548.112,A -85,B 0,C 180,E1 -9812.848,E2 -9812.848} C_VEL
LIN {X 0,Y 424.403,Z 546.626,A -85,B 0,C 180,E1 -9813.798,E2 -9813.798} C_VEL
LIN {X 0,Y 424.349,Z 543.502,A -85,B 0,C 180,E1 -9815.226,E2 -9815.226} C_VEL
LIN {X 0,Y 424.399,Z 539.275,A -85,B 0,C 180,E1 -9816.657,E2 -9816.657} C_VEL
LIN {X 0,Y 424.533,Z 532.782,A -85,B 0,C 180,E1 -9818.329,E2 -9818.329} C_VEL
LIN {X 0,Y 424.77,Z 525.706,A -85,B 0,C 180,E1 -9819.764,E2 -9819.764} C_VEL
LIN {X 0,Y 425.232,Z 516.818,A -85,B 0,C 180,E1 -9821.198,E2 -9821.198} C_VEL
LIN {X 0,Y 425.727,Z 507.724,A -85,B 0,C 180,E1 -9822.393,E2 -9822.393} C_VEL
LIN {X 0,Y 426.249,Z 498.434,A -85,B 0,C 180,E1 -9823.395,E2 -9823.395} C_VEL
LIN {X 0,Y 426.822,Z 488.137,A -85,B 0,C 180,E1 -9824.299,E2 -9824.299} C_VEL
LIN {X 0,Y 427.529,Z 476.133,A -85,B 0,C 180,E1 -9825.127,E2 -9825.127} C_VEL
LIN {X 0,Y 427.825,Z 466.224,A -85,B 0,C 180,E1 -9825.666,E2 -9825.666} C_VEL
LIN {X 0,Y 426.9,Z 453.192,A -85,B 0,C 180,E1 -9826.237,E2 -9826.237} C_VEL
LIN {X 0,Y 425.53,Z 442.889,A -85,B 0,C 180,E1 -9826.587,E2 -9826.587} C_VEL
LIN {X 0,Y 426.488,Z 427.193,A -85,B 0,C 180,E1 -9830.246,E2 -9830.246} C_VEL
LIN {X 0,Y 427.515,Z 415.059,A -85,B 0,C 180,E1 -9833.237,E2 -9833.237} C_VEL
LIN {X 0,Y 428.892,Z 403.539,A -85,B 0,C 180,E1 -9836.259,E2 -9836.259} C_VEL
LIN {X 0,Y 430.38,Z 394.562,A -85,B 0,C 180,E1 -9838.799,E2 -9838.799} C_VEL
LIN {X 0,Y 430.645,Z 391.662,A -85,B 0,C 180,E1 -9839.701,E2 -9839.701} C_VEL
LIN {X 0,Y 429.679,Z 386.077,A -85,B 0,C 180,E1 -9841.73,E2 -9841.73} C_VEL
LIN {X 0,Y 428.632,Z 380.957,A -85,B 0,C 180,E1 -9843.882,E2 -9843.882} C_VEL
LIN {X 0,Y 427.401,Z 376.198,A -85,B 0,C 180,E1 -9846.318,E2 -9846.318} C_VEL
LIN {X 0,Y 426.391,Z 371.868,A -85,B 0,C 180,E1 -9849.224,E2 -9849.224} C_VEL
LIN {X 0,Y 425.723,Z 369.123,A -85,B 0,C 180,E1 -9852.023,E2 -9852.023} C_VEL
LIN {X 0,Y 425.324,Z 367.823,A -85,B 0,C 180,E1 -9854.722,E2 -9854.722} C_VEL
LIN {X 0,Y 425.306,Z 367.673,A -85,B 0,C 180,E1 -9857.351,E2 -9857.351} C_VEL
LIN {X 0,Y 425.528,Z 368.485,A -85,B 0,C 180,E1 -9859.9,E2 -9859.9} C_VEL
LIN {X 0,Y 425.853,Z 370.09,A -85,B 0,C 180,E1 -9862.388,E2 -9862.388} C_VEL
LIN {X 0,Y 426.422,Z 372.95,A -85,B 0,C 180,E1 -9865.494,E2 -9865.494} C_VEL
LIN {X 0,Y 426.886,Z 376.122,A -85,B 0,C 180,E1 -9868.208,E2 -9868.208} C_VEL
LIN {X 0,Y 426.915,Z 379.112,A -85,B 0,C 180,E1 -9870.405,E2 -9870.405} C_VEL
LIN {X 0,Y 426.486,Z 383.957,A -85,B 0,C 180,E1 -9873.581,E2 -9873.581} C_VEL
LIN {X 0,Y 426.062,Z 388.971,A -85,B 0,C 180,E1 -9876.679,E2 -9876.679} C_VEL
LIN {X 0,Y 425.721,Z 395.032,A -85,B 0,C 180,E1 -9880.218,E2 -9880.218} C_VEL
LIN {X 0,Y 425.419,Z 401.222,A -85,B 0,C 180,E1 -9883.689,E2 -9883.689} C_VEL
LIN {X 0,Y 425.143,Z 408.414,A -85,B 0,C 180,E1 -9887.59,E2 -9887.59} C_VEL
LIN {X 0,Y 424.936,Z 411.1,A -85,B 0,C 180,E1 -9889.006,E2 -9889.006} C_VEL
LIN {X 0,Y 427.117,Z 421.341,A -85,B 0,C 180,E1 -9889.692,E2 -9889.692} C_VEL
LIN {X 0,Y 427.452,Z 426.276,A -85,B 0,C 180,E1 -9890.059,E2 -9890.059} C_VEL
LIN {X 0,Y 426.916,Z 436.17,A -85,B 0,C 180,E1 -9890.913,E2 -9890.913} C_VEL
LIN {X 0,Y 426.471,Z 444.159,A -85,B 0,C 180,E1 -9891.811,E2 -9891.811} C_VEL
LIN {X 0,Y 425.958,Z 451.717,A -85,B 0,C 180,E1 -9892.892,E2 -9892.892} C_VEL
LIN {X 0,Y 425.562,Z 458.042,A -85,B 0,C 180,E1 -9894.076,E2 -9894.076} C_VEL
LIN {X 0,Y 425.176,Z 462.819,A -85,B 0,C 180,E1 -9895.259,E2 -9895.259} C_VEL
LIN {X 0,Y 424.926,Z 465.675,A -85,B 0,C 180,E1 -9896.207,E2 -9896.207} C_VEL
LIN {X 0,Y 424.663,Z 467.783,A -85,B 0,C 180,E1 -9897.154,E2 -9897.154} C_VEL
LIN {X 0,Y 424.512,Z 469.178,A -85,B 0,C 180,E1 -9898.103,E2 -9898.103} C_VEL
LIN {X 0,Y 424.43,Z 469.894,A -85,B 0,C 180,E1 -9899.051,E2 -9899.051} C_VEL
LIN {X 0,Y 424.385,Z 469.946,A -85,B 0,C 180,E1 -9900,E2 -9900} C_VEL
LIN {X 0,Y 424.371,Z 469.329,A -85,B 0,C 180,E1 -9900.949,E2 -9900.949} C_VEL
LIN {X 0,Y 424.504,Z 467.124,A -85,B 0,C 180,E1 -9902.372,E2 -9902.372} C_VEL
LIN {X 0,Y 424.804,Z 463.28,A -85,B 0,C 180,E1 -9903.795,E2 -9903.795} C_VEL
LIN {X 0,Y 425.006,Z 458.692,A -85,B 0,C 180,E1 -9904.981,E2 -9904.981} C_VEL
LIN {X 0,Y 425.236,Z 452.571,A -85,B 0,C 180,E1 -9906.167,E2 -9906.167} C_VEL
LIN {X 0,Y 425.365,Z 445.336,A -85,B 0,C 180,E1 -9907.247,E2 -9907.247} C_VEL
LIN {X 0,Y 425.691,Z 437.573,A -85,B 0,C 180,E1 -9908.151,E2 -9908.151} C_VEL
LIN {X 0,Y 426.04,Z 427.922,A -85,B 0,C 180,E1 -9909.016,E2 -9909.016} C_VEL
LIN {X 0,Y 426.081,Z 419.271,A -85,B 0,C 180,E1 -9909.614,E2 -9909.614} C_VEL
LIN {X 0,Y 424.406,Z 408.101,A -85,B 0,C 180,E1 -9910.224,E2 -9910.224} C_VEL
LIN {X 0,Y 424.559,Z 403.555,A -85,B 0,C 180,E1 -9912.427,E2 -9912.427} C_VEL
LIN {X 0,Y 424.73,Z 395.628,A -85,B 0,C 180,E1 -9916.338,E2 -9916.338} C_VEL
LIN {X 0,Y 424.876,Z 389.407,A -85,B 0,C 180,E1 -9919.463,E2 -9919.463} C_VEL
LIN {X 0,Y 425.004,Z 382.72,A -85,B 0,C 180,E1 -9922.868,E2 -9922.868} C_VEL
LIN {X 0,Y 425.201,Z 376.703,A -85,B 0,C 180,E1 -9925.977,E2 -9925.977} C_VEL
LIN {X 0,Y 425.547,Z 369.621,A -85,B 0,C 180,E1 -9929.7,E2 -9929.7} C_VEL
LIN {X 0,Y 425.426,Z 367.495,A -85,B 0,C 180,E1 -9930.943,E2 -9930.943} C_VEL
LIN {X 0,Y 425.315,Z 367.505,A -85,B 0,C 180,E1 -9934.288,E2 -9934.288} C_VEL
LIN {X 0,Y 425.289,Z 367.509,A -85,B 0,C 180,E1 -9937.694,E2 -9937.694} C_VEL
LIN {X 0,Y 425.285,Z 367.51,A -85,B 0,C 180,E1 -9940.521,E2 -9940.521} C_VEL
LIN {X 0,Y 425.261,Z 367.511,A -85,B 0,C 180,E1 -9943.351,E2 -9943.351} C_VEL
LIN {X 0,Y 425.267,Z 367.514,A -85,B 0,C 180,E1 -9946.648,E2 -9946.648} C_VEL
LIN {X 0,Y 425.29,Z 367.509,A -85,B 0,C 180,E1 -9949.873,E2 -9949.873} C_VEL
LIN {X 0,Y 425.281,Z 367.511,A -85,B 0,C 180,E1 -9952.488,E2 -9952.488} C_VEL
LIN {X 0,Y 425.311,Z 367.505,A -85,B 0,C 180,E1 -9955.817,E2 -9955.817} C_VEL
LIN {X 0,Y 425.294,Z 367.509,A -85,B 0,C 180,E1 -9959.239,E2 -9959.239} C_VEL
LIN {X 0,Y 425.353,Z 367.502,A -85,B 0,C 180,E1 -9962.442,E2 -9962.442} C_VEL
LIN {X 0,Y 425.351,Z 367.499,A -85,B 0,C 180,E1 -9965.602,E2 -9965.602} C_VEL
LIN {X 0,Y 425.297,Z 367.508,A -85,B 0,C 180,E1 -9968.682,E2 -9968.682} C_VEL
LIN {X 0,Y 425.337,Z 367.504,A -85,B 0,C 180,E1 -9971.703,E2 -9971.703} C_VEL
LIN {X 0,Y 425.352,Z 367.502,A -85,B 0,C 180,E1 -9974.671,E2 -9974.671} C_VEL
LIN {X 0,Y 425.416,Z 367.492,A -85,B 0,C 180,E1 -9977.598,E2 -9977.598} C_VEL
LIN {X 0,Y 425.446,Z 367.49,A -85,B 0,C 180,E1 -9981.45,E2 -9981.45} C_VEL
LIN {X 0,Y 425.554,Z 367.478,A -85,B 0,C 180,E1 -9984.313,E2 -9984.313} C_VEL
LIN {X 0,Y 425.577,Z 367.476,A -85,B 0,C 180,E1 -9988.107,E2 -9988.107} C_VEL
LIN {X 0,Y 425.706,Z 367.459,A -85,B 0,C 180,E1 -9990,E2 -9990} C_VEL
LIN {X 0,Y 425.56,Z 367.475,A -85,B 0,C 180,E1 -9992.84,E2 -9992.84} C_VEL
LIN {X 0,Y 425.527,Z 367.479,A -85,B 0,C 180,E1 -9996.639,E2 -9996.639} C_VEL
LIN {X 0,Y 425.454,Z 367.486,A -85,B 0,C 180,E1 -9998.328,E2 -9998.328} C_VEL
LIN {X 0,Y 424.75,Z 367.575,A -85,B 0,C 180,E1 -9999.117,E2 -9999.117} C_VEL
LIN {X 0,Y 421.834,Z 367.939,A -85,B 0,C 180,E1 -10000.399,E2 -10000.399} C_VEL
LIN {X 0,Y 419.409,Z 368.243,A -85,B 0,C 180,E1 -10001.434,E2 -10001.434} C_VEL
LIN {X 0,Y 418.409,Z 368.366,A -85,B 0,C 180,E1 -10002.234,E2 -10002.234} C_VEL
LIN {X 0,Y 418.349,Z 368.373,A -85,B 0,C 180,E1 -10002.505,E2 -10002.505} C_VEL
LIN {X 0,Y 418.306,Z 368.38,A -85,B 0,C 180,E1 -10005.594,E2 -10005.594} C_VEL
LIN {X 0,Y 418.288,Z 368.379,A -85,B 0,C 180,E1 -10008.617,E2 -10008.617} C_VEL
LIN {X 0,Y 418.238,Z 368.389,A -85,B 0,C 180,E1 -10011.696,E2 -10011.696} C_VEL
LIN {X 0,Y 418.287,Z 368.381,A -85,B 0,C 180,E1 -10014.864,E2 -10014.864} C_VEL
LIN {X 0,Y 418.295,Z 368.381,A -85,B 0,C 180,E1 -10018.063,E2 -10018.063} C_VEL
LIN {X 0,Y 418.215,Z 368.393,A -85,B 0,C 180,E1 -10021.396,E2 -10021.396} C_VEL
LIN {X 0,Y 418.268,Z 368.383,A -85,B 0,C 180,E1 -10024.58,E2 -10024.58} C_VEL
LIN {X 0,Y 418.232,Z 368.39,A -85,B 0,C 180,E1 -10027.834,E2 -10027.834} C_VEL
LIN {X 0,Y 418.226,Z 368.389,A -85,B 0,C 180,E1 -10030.948,E2 -10030.948} C_VEL
LIN {X 0,Y 418.212,Z 368.39,A -85,B 0,C 180,E1 -10033.729,E2 -10033.729} C_VEL
LIN {X 0,Y 418.211,Z 368.391,A -85,B 0,C 180,E1 -10036.449,E2 -10036.449} C_VEL
LIN {X 0,Y 418.225,Z 368.39,A -85,B 0,C 180,E1 -10039.13,E2 -10039.13} C_VEL
LIN {X 0,Y 418.23,Z 368.386,A -85,B 0,C 180,E1 -10042.167,E2 -10042.167} C_VEL
LIN {X 0,Y 418.268,Z 368.384,A -85,B 0,C 180,E1 -10045.42,E2 -10045.42} C_VEL
LIN {X 0,Y 418.214,Z 368.392,A -85,B 0,C 180,E1 -10048.604,E2 -10048.604} C_VEL
LIN {X 0,Y 418.294,Z 368.379,A -85,B 0,C 180,E1 -10051.937,E2 -10051.937} C_VEL
LIN {X 0,Y 418.292,Z 368.381,A -85,B 0,C 180,E1 -10055.163,E2 -10055.163} C_VEL
LIN {X 0,Y 418.237,Z 368.388,A -85,B 0,C 180,E1 -10058.304,E2 -10058.304} C_VEL
LIN {X 0,Y 418.287,Z 368.382,A -85,B 0,C 180,E1 -10061.383,E2 -10061.383} C_VEL
LIN {X 0,Y 418.305,Z 368.379,A -85,B 0,C 180,E1 -10064.406,E2 -10064.406} C_VEL
LIN {X 0,Y 418.373,Z 368.37,A -85,B 0,C 180,E1 -10067.386,E2 -10067.386} C_VEL
LIN {X 0,Y 418.362,Z 368.373,A -85,B 0,C 180,E1 -10070.329,E2 -10070.329} C_VEL
LIN {X 0,Y 418.497,Z 368.355,A -85,B 0,C 180,E1 -10073.249,E2 -10073.249} C_VEL
LIN {X 0,Y 418.34,Z 368.373,A -85,B 0,C 180,E1 -10075.181,E2 -10075.181} C_VEL
LIN {X 0,Y 418.545,Z 368.35,A -85,B 0,C 180,E1 -10078.075,E2 -10078.075} C_VEL
LIN {X 0,Y 418.676,Z 368.334,A -85,B 0,C 180,E1 -10080,E2 -10080} C_VEL
LIN {X 0,Y 418.513,Z 368.355,A -85,B 0,C 180,E1 -10082.888,E2 -10082.888} C_VEL
LIN {X 0,Y 418.496,Z 368.355,A -85,B 0,C 180,E1 -10086.751,E2 -10086.751} C_VEL
LIN {X 0,Y 418.402,Z 368.367,A -85,B 0,C 180,E1 -10088.695,E2 -10088.695} C_VEL
LIN {X 0,Y 418.318,Z 368.378,A -85,B 0,C 180,E1 -10091.631,E2 -10091.631} C_VEL
LIN {X 0,Y 418.305,Z 368.381,A -85,B 0,C 180,E1 -10094.597,E2 -10094.597} C_VEL
LIN {X 0,Y 418.288,Z 368.38,A -85,B 0,C 180,E1 -10097.604,E2 -10097.604} C_VEL
LIN {X 0,Y 418.252,Z 368.386,A -85,B 0,C 180,E1 -10100.663,E2 -10100.663} C_VEL
LIN {X 0,Y 418.29,Z 368.382,A -85,B 0,C 180,E1 -10103.781,E2 -10103.781} C_VEL
LIN {X 0,Y 418.312,Z 368.377,A -85,B 0,C 180,E1 -10107.07,E2 -10107.07} C_VEL
LIN {X 0,Y 418.246,Z 368.387,A -85,B 0,C 180,E1 -10110.272,E2 -10110.272} C_VEL
LIN {X 0,Y 418.251,Z 368.387,A -85,B 0,C 180,E1 -10113.677,E2 -10113.677} C_VEL
LIN {X 0,Y 418.248,Z 368.386,A -85,B 0,C 180,E1 -10117.223,E2 -10117.223} C_VEL
LIN {X 0,Y 418.257,Z 368.387,A -85,B 0,C 180,E1 -10119.681,E2 -10119.681} C_VEL
LIN {X 0,Y 418.234,Z 368.388,A -85,B 0,C 180,E1 -10122.322,E2 -10122.322} C_VEL
LIN {X 0,Y 418.244,Z 368.387,A -85,B 0,C 180,E1 -10125.11,E2 -10125.11} C_VEL
LIN {X 0,Y 418.244,Z 368.388,A -85,B 0,C 180,E1 -10127.767,E2 -10127.767} C_VEL
LIN {X 0,Y 418.249,Z 368.386,A -85,B 0,C 180,E1 -10131.558,E2 -10131.558} C_VEL
LIN {X 0,Y 418.287,Z 368.469,A -85,B 0,C 180,E1 -10134.794,E2 -10134.794} C_VEL
LIN {X 0,Y 420.739,Z 380.053,A -85,B 0,C 180,E1 -10138.087,E2 -10138.087} C_VEL
LIN {X 0,Y 422.418,Z 388.244,A -85,B 0,C 180,E1 -10140.332,E2 -10140.332} C_VEL
LIN {X 0,Y 422.498,Z 391.455,A -85,B 0,C 180,E1 -10141.158,E2 -10141.158} C_VEL
LIN {X 0,Y 420.95,Z 406.416,A -85,B 0,C 180,E1 -10144.816,E2 -10144.816} C_VEL
LIN {X 0,Y 419.791,Z 420.234,A -85,B 0,C 180,E1 -10148.13,E2 -10148.13} C_VEL
LIN {X 0,Y 418.831,Z 435.171,A -85,B 0,C 180,E1 -10151.662,E2 -10151.662} C_VEL
LIN {X 0,Y 418.35,Z 443.714,A -85,B 0,C 180,E1 -10153.657,E2 -10153.657} C_VEL
LIN {X 0,Y 419.844,Z 459.793,A -85,B 0,C 180,E1 -10154.185,E2 -10154.185} C_VEL
LIN {X 0,Y 420.421,Z 469.022,A -85,B 0,C 180,E1 -10154.611,E2 -10154.611} C_VEL
LIN {X 0,Y 419.907,Z 481.429,A -85,B 0,C 180,E1 -10155.336,E2 -10155.336} C_VEL
LIN {X 0,Y 419.284,Z 493.926,A -85,B 0,C 180,E1 -10156.305,E2 -10156.305} C_VEL
LIN {X 0,Y 418.862,Z 503.163,A -85,B 0,C 180,E1 -10157.208,E2 -10157.208} C_VEL
LIN {X 0,Y 418.305,Z 512.825,A -85,B 0,C 180,E1 -10158.369,E2 -10158.369} C_VEL
LIN {X 0,Y 417.822,Z 521.072,A -85,B 0,C 180,E1 -10159.582,E2 -10159.582} C_VEL
LIN {X 0,Y 417.515,Z 529.123,A -85,B 0,C 180,E1 -10161.042,E2 -10161.042} C_VEL
LIN {X 0,Y 417.38,Z 534.528,A -85,B 0,C 180,E1 -10162.258,E2 -10162.258} C_VEL
LIN {X 0,Y 417.273,Z 539.295,A -85,B 0,C 180,E1 -10163.577,E2 -10163.577} C_VEL
LIN {X 0,Y 417.219,Z 543.713,A -85,B 0,C 180,E1 -10165.169,E2 -10165.169} C_VEL
LIN {X 0,Y 417.337,Z 545.734,A -85,B 0,C 180,E1 -10166.138,E2 -10166.138} C_VEL
LIN {X 0,Y 417.41,Z 547.312,A -85,B 0,C 180,E1 -10167.105,E2 -10167.105} C_VEL
LIN {X 0,Y 417.321,Z 548.418,A -85,B 0,C 180,E1 -10168.07,E2 -10168.07} C_VEL
LIN {X 0,Y 417.23,Z 549.065,A -85,B 0,C 180,E1 -10169.035,E2 -10169.035} C_VEL
LIN {X 0,Y 417.217,Z 549.31,A -85,B 0,C 180,E1 -10170,E2 -10170} C_VEL
LIN {X 0,Y 417.232,Z 549.139,A -85,B 0,C 180,E1 -10170.965,E2 -10170.965} C_VEL
LIN {X 0,Y 417.321,Z 548.508,A -85,B 0,C 180,E1 -10171.93,E2 -10171.93} C_VEL
LIN {X 0,Y 417.351,Z 547.459,A -85,B 0,C 180,E1 -10172.896,E2 -10172.896} C_VEL
LIN {X 0,Y 417.305,Z 545.984,A -85,B 0,C 180,E1 -10173.863,E2 -10173.863} C_VEL
LIN {X 0,Y 417.286,Z 542.883,A -85,B 0,C 180,E1 -10175.315,E2 -10175.315} C_VEL
LIN {X 0,Y 417.32,Z 538.677,A -85,B 0,C 180,E1 -10176.77,E2 -10176.77} C_VEL
LIN {X 0,Y 417.47,Z 532.203,A -85,B 0,C 180,E1 -10178.471,E2 -10178.471} C_VEL
LIN {X 0,Y 417.699,Z 525.157,A -85,B 0,C 180,E1 -10179.931,E2 -10179.931} C_VEL
LIN {X 0,Y 418.22,Z 516.324,A -85,B 0,C 180,E1 -10181.388,E2 -10181.388} C_VEL
LIN {X 0,Y 418.753,Z 507.266,A -85,B 0,C 180,E1 -10182.602,E2 -10182.602} C_VEL
LIN {X 0,Y 419.38,Z 497.329,A -85,B 0,C 180,E1 -10183.692,E2 -10183.692} C_VEL
LIN {X 0,Y 420.036,Z 486.3,A -85,B 0,C 180,E1 -10184.659,E2 -10184.659} C_VEL
LIN {X 0,Y 420.8,Z 474.04,A -85,B 0,C 180,E1 -10185.499,E2 -10185.499} C_VEL
LIN {X 0,Y 420.906,Z 466.236,A -85,B 0,C 180,E1 -10185.93,E2 -10185.93} C_VEL
LIN {X 0,Y 419.981,Z 452.791,A -85,B 0,C 180,E1 -10186.543,E2 -10186.543} C_VEL
LIN {X 0,Y 418.568,Z 442.593,A -85,B 0,C 180,E1 -10186.898,E2 -10186.898} C_VEL
LIN {X 0,Y 419.489,Z 428.579,A -85,B 0,C 180,E1 -10190.247,E2 -10190.247} C_VEL
LIN {X 0,Y 420.484,Z 416.96,A -85,B 0,C 180,E1 -10193.179,E2 -10193.179} C_VEL
LIN {X 0,Y 421.949,Z 405.689,A -85,B 0,C 180,E1 -10196.207,E2 -10196.207} C_VEL
LIN {X 0,Y 423.467,Z 396.791,A -85,B 0,C 180,E1 -10198.77,E2 -10198.77} C_VEL
LIN {X 0,Y 423.854,Z 393.457,A -85,B 0,C 180,E1 -10199.831,E2 -10199.831} C_VEL
LIN {X 0,Y 422.796,Z 387.391,A -85,B 0,C 180,E1 -10202.136,E2 -10202.136} C_VEL
LIN {X 0,Y 421.65,Z 382.06,A -85,B 0,C 180,E1 -10204.521,E2 -10204.521} C_VEL
LIN {X 0,Y 420.458,Z 377.613,A -85,B 0,C 180,E1 -10206.995,E2 -10206.995} C_VEL
LIN {X 0,Y 419.666,Z 373.983,A -85,B 0,C 180,E1 -10209.615,E2 -10209.615} C_VEL
LIN {X 0,Y 419.021,Z 371.444,A -85,B 0,C 180,E1 -10212.44,E2 -10212.44} C_VEL
LIN {X 0,Y 418.7,Z 370.261,A -85,B 0,C 180,E1 -10215.172,E2 -10215.172} C_VEL
LIN {X 0,Y 418.676,Z 370.204,A -85,B 0,C 180,E1 -10217.821,E2 -10217.821} C_VEL
LIN {X 0,Y 418.895,Z 371.153,A -85,B 0,C 180,E1 -10220.513,E2 -10220.513} C_VEL
LIN {X 0,Y 419.27,Z 373.243,A -85,B 0,C 180,E1 -10223.572,E2 -10223.572} C_VEL
LIN {X 0,Y 419.8,Z 376.021,A -85,B 0,C 180,E1 -10226.464,E2 -10226.464} C_VEL
LIN {X 0,Y 420.096,Z 378.724,A -85,B 0,C 180,E1 -10228.761,E2 -10228.761} C_VEL
LIN {X 0,Y 419.944,Z 381.695,A -85,B 0,C 180,E1 -10230.966,E2 -10230.966} C_VEL
LIN {X 0,Y 419.458,Z 386.529,A -85,B 0,C 180,E1 -10234.175,E2 -10234.175} C_VEL
LIN {X 0,Y 419.061,Z 391.546,A -85,B 0,C 180,E1 -10237.311,E2 -10237.311} C_VEL
LIN {X 0,Y 418.72,Z 396.726,A -85,B 0,C 180,E1 -10240.386,E2 -10240.386} C_VEL
LIN {X 0,Y 418.454,Z 401.997,A -85,B 0,C 180,E1 -10243.41,E2 -10243.41} C_VEL
LIN {X 0,Y 418.155,Z 409.172,A -85,B 0,C 180,E1 -10247.379,E2 -10247.379} C_VEL
LIN {X 0,Y 417.95,Z 411.578,A -85,B 0,C 180,E1 -10248.666,E2 -10248.666} C_VEL
LIN {X 0,Y 420.487,Z 423.587,A -85,B 0,C 180,E1 -10249.527,E2 -10249.527} C_VEL
LIN {X 0,Y 420.607,Z 428.321,A -85,B 0,C 180,E1 -10249.895,E2 -10249.895} C_VEL
LIN {X 0,Y 420.119,Z 436.631,A -85,B 0,C 180,E1 -10250.637,E2 -10250.637} C_VEL
LIN {X 0,Y 419.607,Z 444.915,A -85,B 0,C 180,E1 -10251.583,E2 -10251.583} C_VEL
LIN {X 0,Y 419.018,Z 452.944,A -85,B 0,C 180,E1 -10252.773,E2 -10252.773} C_VEL
LIN {X 0,Y 418.578,Z 459.109,A -85,B 0,C 180,E1 -10253.976,E2 -10253.976} C_VEL
LIN {X 0,Y 418.166,Z 463.771,A -85,B 0,C 180,E1 -10255.18,E2 -10255.18} C_VEL
LIN {X 0,Y 417.899,Z 466.572,A -85,B 0,C 180,E1 -10256.143,E2 -10256.143} C_VEL
LIN {X 0,Y 417.623,Z 468.63,A -85,B 0,C 180,E1 -10257.106,E2 -10257.106} C_VEL
LIN {X 0,Y 417.461,Z 469.975,A -85,B 0,C 180,E1 -10258.071,E2 -10258.071} C_VEL
LIN {X 0,Y 417.371,Z 470.641,A -85,B 0,C 180,E1 -10259.035,E2 -10259.035} C_VEL
LIN {X 0,Y 417.32,Z 470.641,A -85,B 0,C 180,E1 -10260,E2 -10260} C_VEL
LIN {X 0,Y 417.309,Z 469.969,A -85,B 0,C 180,E1 -10260.965,E2 -10260.965} C_VEL
LIN {X 0,Y 417.45,Z 467.68,A -85,B 0,C 180,E1 -10262.412,E2 -10262.412} C_VEL
LIN {X 0,Y 417.747,Z 463.758,A -85,B 0,C 180,E1 -10263.859,E2 -10263.859} C_VEL
LIN {X 0,Y 417.965,Z 459.097,A -85,B 0,C 180,E1 -10265.065,E2 -10265.065} C_VEL
LIN {X 0,Y 418.179,Z 452.907,A -85,B 0,C 180,E1 -10266.272,E2 -10266.272} C_VEL
LIN {X 0,Y 418.328,Z 446.144,A -85,B 0,C 180,E1 -10267.299,E2 -10267.299} C_VEL
LIN {X 0,Y 418.684,Z 437.425,A -85,B 0,C 180,E1 -10268.325,E2 -10268.325} C_VEL
LIN {X 0,Y 419.035,Z 428.057,A -85,B 0,C 180,E1 -10269.168,E2 -10269.168} C_VEL
LIN {X 0,Y 419.162,Z 421.261,A -85,B 0,C 180,E1 -10269.652,E2 -10269.652} C_VEL
LIN {X 0,Y 417.718,Z 411.269,A -85,B 0,C 180,E1 -10270.237,E2 -10270.237} C_VEL
LIN {X 0,Y 417.339,Z 408.335,A -85,B 0,C 180,E1 -10270.399,E2 -10270.399} C_VEL
LIN {X 0,Y 417.476,Z 403.758,A -85,B 0,C 180,E1 -10272.642,E2 -10272.642} C_VEL
LIN {X 0,Y 417.663,Z 395.77,A -85,B 0,C 180,E1 -10276.622,E2 -10276.622} C_VEL
LIN {X 0,Y 417.847,Z 388.796,A -85,B 0,C 180,E1 -10280.17,E2 -10280.17} C_VEL
LIN {X 0,Y 417.979,Z 382.787,A -85,B 0,C 180,E1 -10283.275,E2 -10283.275} C_VEL
LIN {X 0,Y 418.208,Z 376.716,A -85,B 0,C 180,E1 -10286.445,E2 -10286.445} C_VEL
LIN {X 0,Y 418.52,Z 370.58,A -85,B 0,C 180,E1 -10289.695,E2 -10289.695} C_VEL
LIN {X 0,Y 418.386,Z 368.372,A -85,B 0,C 180,E1 -10290.962,E2 -10290.962} C_VEL
LIN {X 0,Y 418.263,Z 368.387,A -85,B 0,C 180,E1 -10294.841,E2 -10294.841} C_VEL
LIN {X 0,Y 418.263,Z 368.386,A -85,B 0,C 180,E1 -10298.441,E2 -10298.441} C_VEL
LIN {X 0,Y 418.226,Z 368.391,A -85,B 0,C 180,E1 -10300.948,E2 -10300.948} C_VEL
LIN {X 0,Y 418.213,Z 368.388,A -85,B 0,C 180,E1 -10303.729,E2 -10303.729} C_VEL
LIN {X 0,Y 418.219,Z 368.392,A -85,B 0,C 180,E1 -10306.45,E2 -10306.45} C_VEL
LIN {X 0,Y 418.226,Z 368.391,A -85,B 0,C 180,E1 -10309.13,E2 -10309.13} C_VEL
LIN {X 0,Y 418.231,Z 368.388,A -85,B 0,C 180,E1 -10312.167,E2 -10312.167} C_VEL
LIN {X 0,Y 418.269,Z 368.381,A -85,B 0,C 180,E1 -10315.42,E2 -10315.42} C_VEL
LIN {X 0,Y 418.215,Z 368.391,A -85,B 0,C 180,E1 -10318.604,E2 -10318.604} C_VEL
LIN {X 0,Y 418.295,Z 368.381,A -85,B 0,C 180,E1 -10321.937,E2 -10321.937} C_VEL
LIN {X 0,Y 418.293,Z 368.378,A -85,B 0,C 180,E1 -10325.163,E2 -10325.163} C_VEL
LIN {X 0,Y 418.238,Z 368.389,A -85,B 0,C 180,E1 -10328.304,E2 -10328.304} C_VEL
LIN {X 0,Y 418.287,Z 368.381,A -85,B 0,C 180,E1 -10331.383,E2 -10331.383} C_VEL
LIN {X 0,Y 418.307,Z 368.382,A -85,B 0,C 180,E1 -10334.406,E2 -10334.406} C_VEL
LIN {X 0,Y 418.359,Z 368.37,A -85,B 0,C 180,E1 -10337.386,E2 -10337.386} C_VEL
LIN {X 0,Y 418.344,Z 368.375,A -85,B 0,C 180,E1 -10340.329,E2 -10340.329} C_VEL
LIN {X 0,Y 418.491,Z 368.355,A -85,B 0,C 180,E1 -10343.249,E2 -10343.249} C_VEL
LIN {X 0,Y 418.342,Z 368.373,A -85,B 0,C 180,E1 -10345.181,E2 -10345.181} C_VEL
LIN {X 0,Y 418.546,Z 368.352,A -85,B 0,C 180,E1 -10348.075,E2 -10348.075} C_VEL
LIN {X 0,Y 418.675,Z 368.335,A -85,B 0,C 180,E1 -10350,E2 -10350} C_VEL
LIN {X 0,Y 418.514,Z 368.353,A -85,B 0,C 180,E1 -10352.888,E2 -10352.888} C_VEL
LIN {X 0,Y 418.491,Z 368.354,A -85,B 0,C 180,E1 -10356.751,E2 -10356.751} C_VEL
LIN {X 0,Y 418.361,Z 368.374,A -85,B 0,C 180,E1 -10359.671,E2 -10359.671} C_VEL
LIN {X 0,Y 418.349,Z 368.373,A -85,B 0,C 180,E1 -10362.505,E2 -10362.505} C_VEL
LIN {X 0,Y 417.722,Z 368.453,A -85,B 0,C 180,E1 -10363.309,E2 -10363.309} C_VEL
LIN {X 0,Y 414.828,Z 368.812,A -85,B 0,C 180,E1 -10364.612,E2 -10364.612} C_VEL
LIN {X 0,Y 412.364,Z 369.12,A -85,B 0,C 180,E1 -10365.665,E2 -10365.665} C_VEL
LIN {X 0,Y 411.329,Z 369.247,A -85,B 0,C 180,E1 -10366.48,E2 -10366.48} C_VEL
LIN {X 0,Y 411.259,Z 369.255,A -85,B 0,C 180,E1 -10366.756,E2 -10366.756} C_VEL
LIN {X 0,Y 411.258,Z 369.257,A -85,B 0,C 180,E1 -10369.985,E2 -10369.985} C_VEL
LIN {X 0,Y 411.206,Z 369.264,A -85,B 0,C 180,E1 -10373.147,E2 -10373.147} C_VEL
LIN {X 0,Y 411.241,Z 369.258,A -85,B 0,C 180,E1 -10376.381,E2 -10376.381} C_VEL
LIN {X 0,Y 411.203,Z 369.266,A -85,B 0,C 180,E1 -10379.712,E2 -10379.712} C_VEL
LIN {X 0,Y 411.209,Z 369.265,A -85,B 0,C 180,E1 -10383.156,E2 -10383.156} C_VEL
LIN {X 0,Y 411.195,Z 369.264,A -85,B 0,C 180,E1 -10386.552,E2 -10386.552} C_VEL
LIN {X 0,Y 411.22,Z 369.262,A -85,B 0,C 180,E1 -10389.729,E2 -10389.729} C_VEL
LIN {X 0,Y 411.176,Z 369.27,A -85,B 0,C 180,E1 -10393.133,E2 -10393.133} C_VEL
LIN {X 0,Y 411.17,Z 369.268,A -85,B 0,C 180,E1 -10395.881,E2 -10395.881} C_VEL
LIN {X 0,Y 411.166,Z 369.269,A -85,B 0,C 180,E1 -10398.772,E2 -10398.772} C_VEL
LIN {X 0,Y 411.196,Z 369.262,A -85,B 0,C 180,E1 -10402.026,E2 -10402.026} C_VEL
LIN {X 0,Y 411.208,Z 369.263,A -85,B 0,C 180,E1 -10405.666,E2 -10405.666} C_VEL
LIN {X 0,Y 411.192,Z 369.267,A -85,B 0,C 180,E1 -10409.152,E2 -10409.152} C_VEL
LIN {X 0,Y 411.261,Z 369.256,A -85,B 0,C 180,E1 -10412.522,E2 -10412.522} C_VEL
LIN {X 0,Y 411.23,Z 369.259,A -85,B 0,C 180,E1 -10415.785,E2 -10415.785} C_VEL
LIN {X 0,Y 411.199,Z 369.265,A -85,B 0,C 180,E1 -10418.966,E2 -10418.966} C_VEL
LIN {X 0,Y 411.255,Z 369.257,A -85,B 0,C 180,E1 -10422.085,E2 -10422.085} C_VEL
LIN {X 0,Y 411.265,Z 369.256,A -85,B 0,C 180,E1 -10425.147,E2 -10425.147} C_VEL
LIN {X 0,Y 411.302,Z 369.252,A -85,B 0,C 180,E1 -10428.168,E2 -10428.168} C_VEL
LIN {X 0,Y 411.484,Z 369.229,A -85,B 0,C 180,E1 -10432.147,E2 -10432.147} C_VEL
LIN {X 0,Y 411.478,Z 369.229,A -85,B 0,C 180,E1 -10434.118,E2 -10434.118} C_VEL
LIN {X 0,Y 411.514,Z 369.225,A -85,B 0,C 180,E1 -10438.042,E2 -10438.042} C_VEL
LIN {X 0,Y 411.645,Z 369.21,A -85,B 0,C 180,E1 -10440,E2 -10440} C_VEL
LIN {X 0,Y 411.468,Z 369.232,A -85,B 0,C 180,E1 -10442.937,E2 -10442.937} C_VEL
LIN {X 0,Y 411.463,Z 369.23,A -85,B 0,C 180,E1 -10446.867,E2 -10446.867} C_VEL
LIN {X 0,Y 411.295,Z 369.253,A -85,B 0,C 180,E1 -10449.839,E2 -10449.839} C_VEL
LIN {X 0,Y 411.308,Z 369.25,A -85,B 0,C 180,E1 -10453.104,E2 -10453.104} C_VEL
LIN {X 0,Y 411.265,Z 369.254,A -85,B 0,C 180,E1 -10456.869,E2 -10456.869} C_VEL
LIN {X 0,Y 411.232,Z 369.263,A -85,B 0,C 180,E1 -10459.987,E2 -10459.987} C_VEL
LIN {X 0,Y 411.205,Z 369.263,A -85,B 0,C 180,E1 -10463.147,E2 -10463.147} C_VEL
LIN {X 0,Y 411.24,Z 369.261,A -85,B 0,C 180,E1 -10466.381,E2 -10466.381} C_VEL
LIN {X 0,Y 411.202,Z 369.265,A -85,B 0,C 180,E1 -10469.713,E2 -10469.713} C_VEL
LIN {X 0,Y 411.208,Z 369.263,A -85,B 0,C 180,E1 -10473.156,E2 -10473.156} C_VEL
LIN {X 0,Y 411.197,Z 369.264,A -85,B 0,C 180,E1 -10476.553,E2 -10476.553} C_VEL
LIN {X 0,Y 411.221,Z 369.264,A -85,B 0,C 180,E1 -10479.729,E2 -10479.729} C_VEL
LIN {X 0,Y 411.18,Z 369.266,A -85,B 0,C 180,E1 -10483.133,E2 -10483.133} C_VEL
LIN {X 0,Y 411.175,Z 369.268,A -85,B 0,C 180,E1 -10485.88,E2 -10485.88} C_VEL
LIN {X 0,Y 411.166,Z 369.267,A -85,B 0,C 180,E1 -10488.772,E2 -10488.772} C_VEL
LIN {X 0,Y 411.193,Z 369.264,A -85,B 0,C 180,E1 -10492.026,E2 -10492.026} C_VEL
LIN {X 0,Y 411.237,Z 369.382,A -85,B 0,C 180,E1 -10494.475,E2 -10494.475} C_VEL
LIN {X 0,Y 413.296,Z 379.124,A -85,B 0,C 180,E1 -10497.323,E2 -10497.323} C_VEL
LIN {X 0,Y 415.42,Z 389.314,A -85,B 0,C 180,E1 -10500.176,E2 -10500.176} C_VEL
LIN {X 0,Y 415.478,Z 393.142,A -85,B 0,C 180,E1 -10501.178,E2 -10501.178} C_VEL
LIN {X 0,Y 413.891,Z 407.986,A -85,B 0,C 180,E1 -10504.88,E2 -10504.88} C_VEL
LIN {X 0,Y 412.61,Z 422.83,A -85,B 0,C 180,E1 -10508.518,E2 -10508.518} C_VEL
LIN {X 0,Y 411.557,Z 438.864,A -85,B 0,C 180,E1 -10512.381,E2 -10512.381} C_VEL
LIN {X 0,Y 411.296,Z 443.538,A -85,B 0,C 180,E1 -10513.496,E2 -10513.496} C_VEL
LIN {X 0,Y 412.528,Z 456.869,A -85,B 0,C 180,E1 -10513.912,E2 -10513.912} C_VEL
LIN {X 0,Y 413.41,Z 469.064,A -85,B 0,C 180,E1 -10514.47,E2 -10514.47} C_VEL
LIN {X 0,Y 412.887,Z 481.308,A -85,B 0,C 180,E1 -10515.207,E2 -10515.207} C_VEL
LIN {X 0,Y 412.251,Z 493.721,A -85,B 0,C 180,E1 -10516.192,E2 -10516.192} C_VEL
LIN {X 0,Y 411.77,Z 503.511,A -85,B 0,C 180,E1 -10517.18,E2 -10517.18} C_VEL
LIN {X 0,Y 411.191,Z 513.396,A -85,B 0,C 180,E1 -10518.415,E2 -10518.415} C_VEL
LIN {X 0,Y 410.704,Z 521.452,A -85,B 0,C 180,E1 -10519.649,E2 -10519.649} C_VEL
LIN {X 0,Y 410.44,Z 529.28,A -85,B 0,C 180,E1 -10521.135,E2 -10521.135} C_VEL
LIN {X 0,Y 410.279,Z 535.476,A -85,B 0,C 180,E1 -10522.619,E2 -10522.619} C_VEL
LIN {X 0,Y 410.208,Z 540.325,A -85,B 0,C 180,E1 -10524.1,E2 -10524.1} C_VEL
LIN {X 0,Y 410.179,Z 543.971,A -85,B 0,C 180,E1 -10525.578,E2 -10525.578} C_VEL
LIN {X 0,Y 410.346,Z 546.545,A -85,B 0,C 180,E1 -10527.055,E2 -10527.055} C_VEL
LIN {X 0,Y 410.272,Z 547.688,A -85,B 0,C 180,E1 -10528.037,E2 -10528.037} C_VEL
LIN {X 0,Y 410.175,Z 548.351,A -85,B 0,C 180,E1 -10529.018,E2 -10529.018} C_VEL
LIN {X 0,Y 410.159,Z 548.61,A -85,B 0,C 180,E1 -10530,E2 -10530} C_VEL
LIN {X 0,Y 410.177,Z 548.461,A -85,B 0,C 180,E1 -10530.982,E2 -10530.982} C_VEL
LIN {X 0,Y 410.269,Z 547.851,A -85,B 0,C 180,E1 -10531.963,E2 -10531.963} C_VEL
LIN {X 0,Y 410.277,Z 546.809,A -85,B 0,C 180,E1 -10532.946,E2 -10532.946} C_VEL
LIN {X 0,Y 410.209,Z 545.345,A -85,B 0,C 180,E1 -10533.93,E2 -10533.93} C_VEL
LIN {X 0,Y 410.197,Z 542.27,A -85,B 0,C 180,E1 -10535.407,E2 -10535.407} C_VEL
LIN {X 0,Y 410.251,Z 538.098,A -85,B 0,C 180,E1 -10536.887,E2 -10536.887} C_VEL
LIN {X 0,Y 410.39,Z 531.653,A -85,B 0,C 180,E1 -10538.618,E2 -10538.618} C_VEL
LIN {X 0,Y 410.645,Z 524.643,A -85,B 0,C 180,E1 -10540.103,E2 -10540.103} C_VEL
LIN {X 0,Y 411.123,Z 517.5,A -85,B 0,C 180,E1 -10541.338,E2 -10541.338} C_VEL
LIN {X 0,Y 411.621,Z 508.84,A -85,B 0,C 180,E1 -10542.574,E2 -10542.574} C_VEL
LIN {X 0,Y 412.354,Z 498.197,A -85,B 0,C 180,E1 -10543.805,E2 -10543.805} C_VEL
LIN {X 0,Y 413.038,Z 487.672,A -85,B 0,C 180,E1 -10544.787,E2 -10544.787} C_VEL
LIN {X 0,Y 413.827,Z 475.957,A -85,B 0,C 180,E1 -10545.641,E2 -10545.641} C_VEL
LIN {X 0,Y 414.114,Z 467.641,A -85,B 0,C 180,E1 -10546.135,E2 -10546.135} C_VEL
LIN {X 0,Y 413.232,Z 453.875,A -85,B 0,C 180,E1 -10546.806,E2 -10546.806} C_VEL
LIN {X 0,Y 411.594,Z 442.198,A -85,B 0,C 180,E1 -10547.251,E2 -10547.251} C_VEL
LIN {X 0,Y 412.591,Z 428.486,A -85,B 0,C 180,E1 -10550.626,E2 -10550.626} C_VEL
LIN {X 0,Y 413.613,Z 417.718,A -85,B 0,C 180,E1 -10553.429,E2 -10553.429} C_VEL
LIN {X 0,Y 415.234,Z 406.074,A -85,B 0,C 180,E1 -10556.649,E2 -10556.649} C_VEL
LIN {X 0,Y 416.853,Z 397.379,A -85,B 0,C 180,E1 -10559.271,E2 -10559.271} C_VEL
LIN {X 0,Y 416.917,Z 394.151,A -85,B 0,C 180,E1 -10560.379,E2 -10560.379} C_VEL
LIN {X 0,Y 415.559,Z 386.95,A -85,B 0,C 180,E1 -10563.343,E2 -10563.343} C_VEL
LIN {X 0,Y 414.534,Z 382.592,A -85,B 0,C 180,E1 -10565.532,E2 -10565.532} C_VEL
LIN {X 0,Y 413.343,Z 377.909,A -85,B 0,C 180,E1 -10568.544,E2 -10568.544} C_VEL
LIN {X 0,Y 412.865,Z 375.842,A -85,B 0,C 180,E1 -10570.305,E2 -10570.305} C_VEL
LIN {X 0,Y 412.281,Z 373.719,A -85,B 0,C 180,E1 -10572.99,E2 -10572.99} C_VEL
LIN {X 0,Y 412.055,Z 372.693,A -85,B 0,C 180,E1 -10575.754,E2 -10575.754} C_VEL
LIN {X 0,Y 412.043,Z 372.832,A -85,B 0,C 180,E1 -10578.633,E2 -10578.633} C_VEL
LIN {X 0,Y 412.279,Z 374.094,A -85,B 0,C 180,E1 -10581.642,E2 -10581.642} C_VEL
LIN {X 0,Y 412.728,Z 376.48,A -85,B 0,C 180,E1 -10584.821,E2 -10584.821} C_VEL
LIN {X 0,Y 413.08,Z 378.639,A -85,B 0,C 180,E1 -10587.014,E2 -10587.014} C_VEL
LIN {X 0,Y 413.22,Z 381.341,A -85,B 0,C 180,E1 -10589.32,E2 -10589.32} C_VEL
LIN {X 0,Y 412.959,Z 384.328,A -85,B 0,C 180,E1 -10591.541,E2 -10591.541} C_VEL
LIN {X 0,Y 412.473,Z 389.1,A -85,B 0,C 180,E1 -10594.788,E2 -10594.788} C_VEL
LIN {X 0,Y 412.009,Z 394.135,A -85,B 0,C 180,E1 -10597.959,E2 -10597.959} C_VEL
LIN {X 0,Y 411.659,Z 399.29,A -85,B 0,C 180,E1 -10601.072,E2 -10601.072} C_VEL
LIN {X 0,Y 411.335,Z 404.577,A -85,B 0,C 180,E1 -10604.135,E2 -10604.135} C_VEL
LIN {X 0,Y 411.143,Z 409.952,A -85,B 0,C 180,E1 -10607.161,E2 -10607.161} C_VEL
LIN {X 0,Y 410.978,Z 412.06,A -85,B 0,C 180,E1 -10608.315,E2 -10608.315} C_VEL
LIN {X 0,Y 413.347,Z 422.702,A -85,B 0,C 180,E1 -10609.097,E2 -10609.097} C_VEL
LIN {X 0,Y 413.947,Z 427.393,A -85,B 0,C 180,E1 -10609.484,E2 -10609.484} C_VEL
LIN {X 0,Y 413.313,Z 437.318,A -85,B 0,C 180,E1 -10610.376,E2 -10610.376} C_VEL
LIN {X 0,Y 412.744,Z 445.873,A -85,B 0,C 180,E1 -10611.376,E2 -10611.376} C_VEL
LIN {X 0,Y 412.2,Z 452.809,A -85,B 0,C 180,E1 -10612.407,E2 -10612.407} C_VEL
LIN {X 0,Y 411.744,Z 459.174,A -85,B 0,C 180,E1 -10613.63,E2 -10613.63} C_VEL
LIN {X 0,Y 411.343,Z 463.136,A -85,B 0,C 180,E1 -10614.608,E2 -10614.608} C_VEL
LIN {X 0,Y 411.156,Z 466.228,A -85,B 0,C 180,E1 -10615.589,E2 -10615.589} C_VEL
LIN {X 0,Y 410.586,Z 469.495,A -85,B 0,C 180,E1 -10617.057,E2 -10617.057} C_VEL
LIN {X 0,Y 410.411,Z 470.774,A -85,B 0,C 180,E1 -10618.037,E2 -10618.037} C_VEL
LIN {X 0,Y 410.312,Z 471.383,A -85,B 0,C 180,E1 -10619.019,E2 -10619.019} C_VEL
LIN {X 0,Y 410.256,Z 471.331,A -85,B 0,C 180,E1 -10620,E2 -10620} C_VEL
LIN {X 0,Y 410.25,Z 470.607,A -85,B 0,C 180,E1 -10620.982,E2 -10620.982} C_VEL
LIN {X 0,Y 410.398,Z 468.233,A -85,B 0,C 180,E1 -10622.454,E2 -10622.454} C_VEL
LIN {X 0,Y 410.693,Z 464.22,A -85,B 0,C 180,E1 -10623.925,E2 -10623.925} C_VEL
LIN {X 0,Y 410.926,Z 459.468,A -85,B 0,C 180,E1 -10625.152,E2 -10625.152} C_VEL
LIN {X 0,Y 411.119,Z 453.179,A -85,B 0,C 180,E1 -10626.38,E2 -10626.38} C_VEL
LIN {X 0,Y 411.301,Z 445.633,A -85,B 0,C 180,E1 -10627.514,E2 -10627.514} C_VEL
LIN {X 0,Y 411.657,Z 437.466,A -85,B 0,C 180,E1 -10628.468,E2 -10628.468} C_VEL
LIN {X 0,Y 412.02,Z 427.983,A -85,B 0,C 180,E1 -10629.326,E2 -10629.326} C_VEL
LIN {X 0,Y 412.071,Z 421.106,A -85,B 0,C 180,E1 -10629.82,E2 -10629.82} C_VEL
LIN {X 0,Y 410.555,Z 410.859,A -85,B 0,C 180,E1 -10630.417,E2 -10630.417} C_VEL
LIN {X 0,Y 410.271,Z 408.625,A -85,B 0,C 180,E1 -10630.549,E2 -10630.549} C_VEL
LIN {X 0,Y 410.396,Z 402.947,A -85,B 0,C 180,E1 -10633.367,E2 -10633.367} C_VEL
LIN {X 0,Y 410.592,Z 395.905,A -85,B 0,C 180,E1 -10636.917,E2 -10636.917} C_VEL
LIN {X 0,Y 410.783,Z 388.868,A -85,B 0,C 180,E1 -10640.532,E2 -10640.532} C_VEL
LIN {X 0,Y 410.946,Z 382.812,A -85,B 0,C 180,E1 -10643.697,E2 -10643.697} C_VEL
